LIN {X 0,Y 514.55,Z 869.976,A -85,B 0,C 180,E1 14915.309,E2 14915.309} C_VEL
LIN {X 0,Y 492.785,Z 832.233,A -85,B 0,C 180,E1 14922.914,E2 14922.914} C_VEL
LIN {X 0,Y 477.304,Z 810.224,A -85,B 0,C 180,E1 14930.14,E2 14930.14} C_VEL
LIN {X 0,Y 468.627,Z 798.013,A -85,B 0,C 180,E1 14937.192,E2 14937.192} C_VEL
LIN {X 0,Y 469.402,Z 798.715,A -85,B 0,C 180,E1 14950.485,E2 14950.485} C_VEL
LIN {X 0,Y 482.559,Z 818.186,A -85,B 0,C 180,E1 14959.5,E2 14959.5} C_VEL
LIN {X 0,Y 502.665,Z 847.975,A -85,B 0,C 180,E1 14967.396,E2 14967.396} C_VEL
LIN {X 0,Y 523.166,Z 888.461,A -85,B 0,C 180,E1 14974.072,E2 14974.072} C_VEL
LIN {X 0,Y 527.877,Z 903.855,A -85,B 0,C 180,E1 14975.873,E2 14975.873} C_VEL
LIN {X 0,Y 512.114,Z 972.966,A -85,B 0,C 180,E1 14979.163,E2 14979.163} C_VEL
LIN {X 0,Y 492.159,Z 1039.607,A -85,B 0,C 180,E1 14984.274,E2 14984.274} C_VEL
LIN {X 0,Y 472.146,Z 1098.486,A -85,B 0,C 180,E1 14991.255,E2 14991.255} C_VEL
LIN {X 0,Y 456.172,Z 1146.776,A -85,B 0,C 180,E1 14999.951,E2 14999.951} C_VEL
LIN {X 0,Y 446.7,Z 1181.826,A -85,B 0,C 180,E1 15009.677,E2 15009.677} C_VEL
LIN {X 0,Y 443.594,Z 1200.387,A -85,B 0,C 180,E1 15018.207,E2 15018.207} C_VEL
LIN {X 0,Y 443.244,Z 1209.25,A -85,B 0,C 180,E1 15027.105,E2 15027.105} C_VEL
LIN {X 0,Y 443.109,Z 1207.059,A -85,B 0,C 180,E1 15036.281,E2 15036.281} C_VEL
LIN {X 0,Y 443.626,Z 1202.099,A -85,B 0,C 180,E1 15040.69,E2 15040.69} C_VEL
LIN {X 0,Y 436.653,Z 1194.823,A -85,B 0,C 180,E1 15045.123,E2 15045.123} C_VEL
LIN {X 0,Y 442.918,Z 1167.046,A -85,B 0,C 180,E1 15055.407,E2 15055.407} C_VEL
LIN {X 0,Y 455.683,Z 1125.539,A -85,B 0,C 180,E1 15064.822,E2 15064.822} C_VEL
LIN {X 0,Y 473.88,Z 1072.19,A -85,B 0,C 180,E1 15072.665,E2 15072.665} C_VEL
LIN {X 0,Y 493.668,Z 1009.04,A -85,B 0,C 180,E1 15078.748,E2 15078.748} C_VEL
LIN {X 0,Y 512.086,Z 936.922,A -85,B 0,C 180,E1 15083.109,E2 15083.109} C_VEL
LIN {X 0,Y 518.041,Z 902.964,A -85,B 0,C 180,E1 15084.593,E2 15084.593} C_VEL
LIN {X 0,Y 491.056,Z 847.52,A -85,B 0,C 180,E1 15092.061,E2 15092.061} C_VEL
LIN {X 0,Y 465.874,Z 809.438,A -85,B 0,C 180,E1 15099.537,E2 15099.537} C_VEL
LIN {X 0,Y 445.387,Z 782.11,A -85,B 0,C 180,E1 15108.144,E2 15108.144} C_VEL
LIN {X 0,Y 438.046,Z 773.763,A -85,B 0,C 180,E1 15112.94,E2 15112.94} C_VEL
LIN {X 0,Y 434.63,Z 767.06,A -85,B 0,C 180,E1 15117.025,E2 15117.025} C_VEL
LIN {X 0,Y 434.603,Z 767.06,A -85,B 0,C 180,E1 15127.044,E2 15127.044} C_VEL
LIN {X 0,Y 434.587,Z 769.596,A -85,B 0,C 180,E1 15130.777,E2 15130.777} C_VEL
LIN {X 0,Y 441.296,Z 778.041,A -85,B 0,C 180,E1 15136.565,E2 15136.565} C_VEL
LIN {X 0,Y 453.228,Z 793.03,A -85,B 0,C 180,E1 15142.813,E2 15142.813} C_VEL
LIN {X 0,Y 476.279,Z 824.499,A -85,B 0,C 180,E1 15150.896,E2 15150.896} C_VEL
LIN {X 0,Y 501.922,Z 869.101,A -85,B 0,C 180,E1 15158.245,E2 15158.245} C_VEL
LIN {X 0,Y 517.004,Z 906.387,A -85,B 0,C 180,E1 15162.841,E2 15162.841} C_VEL
LIN {X 0,Y 500.153,Z 980.626,A -85,B 0,C 180,E1 15166.741,E2 15166.741} C_VEL
LIN {X 0,Y 480.671,Z 1045.404,A -85,B 0,C 180,E1 15172.189,E2 15172.189} C_VEL
LIN {X 0,Y 461.137,Z 1102.24,A -85,B 0,C 180,E1 15179.556,E2 15179.556} C_VEL
LIN {X 0,Y 446.003,Z 1147.052,A -85,B 0,C 180,E1 15188.497,E2 15188.497} C_VEL
LIN {X 0,Y 438.075,Z 1177.151,A -85,B 0,C 180,E1 15197.956,E2 15197.956} C_VEL
LIN {X 0,Y 435.754,Z 1194.997,A -85,B 0,C 180,E1 15207.955,E2 15207.955} C_VEL
LIN {X 0,Y 434.823,Z 1200.244,A -85,B 0,C 180,E1 15216.965,E2 15216.965} C_VEL
LIN {X 0,Y 435.396,Z 1194.315,A -85,B 0,C 180,E1 15226.549,E2 15226.549} C_VEL
LIN {X 0,Y 438.157,Z 1176.862,A -85,B 0,C 180,E1 15236.071,E2 15236.071} C_VEL
LIN {X 0,Y 446.753,Z 1145.298,A -85,B 0,C 180,E1 15245.895,E2 15245.895} C_VEL
LIN {X 0,Y 462.863,Z 1099.022,A -85,B 0,C 180,E1 15255.059,E2 15255.059} C_VEL
LIN {X 0,Y 484.058,Z 1040.692,A -85,B 0,C 180,E1 15262.524,E2 15262.524} C_VEL
LIN {X 0,Y 504.988,Z 975.634,A -85,B 0,C 180,E1 15267.875,E2 15267.875} C_VEL
LIN {X 0,Y 521.46,Z 903.347,A -85,B 0,C 180,E1 15271.757,E2 15271.757} C_VEL
LIN {X 0,Y 504.014,Z 862.678,A -85,B 0,C 180,E1 15278.05,E2 15278.05} C_VEL
LIN {X 0,Y 482.677,Z 826.981,A -85,B 0,C 180,E1 15286.689,E2 15286.689} C_VEL
LIN {X 0,Y 471.37,Z 812.429,A -85,B 0,C 180,E1 15293.352,E2 15293.352} C_VEL
LIN {X 0,Y 466.641,Z 805.604,A -85,B 0,C 180,E1 15298.473,E2 15298.473} C_VEL
LIN {X 0,Y 468.304,Z 806.975,A -85,B 0,C 180,E1 15310.415,E2 15310.415} C_VEL
LIN {X 0,Y 480.553,Z 825.384,A -85,B 0,C 180,E1 15319.13,E2 15319.13} C_VEL
LIN {X 0,Y 500.058,Z 855.303,A -85,B 0,C 180,E1 15327.161,E2 15327.161} C_VEL
LIN {X 0,Y 519.378,Z 895.393,A -85,B 0,C 180,E1 15333.839,E2 15333.839} C_VEL
LIN {X 0,Y 522.432,Z 908.933,A -85,B 0,C 180,E1 15335.312,E2 15335.312} C_VEL
LIN {X 0,Y 504.887,Z 981.045,A -85,B 0,C 180,E1 15338.924,E2 15338.924} C_VEL
LIN {X 0,Y 483.99,Z 1046.888,A -85,B 0,C 180,E1 15344.271,E2 15344.271} C_VEL
LIN {X 0,Y 463.175,Z 1105.249,A -85,B 0,C 180,E1 15351.62,E2 15351.62} C_VEL
LIN {X 0,Y 447.239,Z 1151.808,A -85,B 0,C 180,E1 15360.588,E2 15360.588} C_VEL
LIN {X 0,Y 438.359,Z 1184.435,A -85,B 0,C 180,E1 15370.329,E2 15370.329} C_VEL
LIN {X 0,Y 435.527,Z 1203.211,A -85,B 0,C 180,E1 15380.019,E2 15380.019} C_VEL
LIN {X 0,Y 434.847,Z 1209.603,A -85,B 0,C 180,E1 15389.05,E2 15389.05} C_VEL
LIN {X 0,Y 435.31,Z 1205.545,A -85,B 0,C 180,E1 15398.064,E2 15398.064} C_VEL
LIN {X 0,Y 436.653,Z 1194.823,A -85,B 0,C 180,E1 15405.123,E2 15405.123} C_VEL
LIN {X 0,Y 430.369,Z 1185.528,A -85,B 0,C 180,E1 15409.593,E2 15409.593} C_VEL
LIN {X 0,Y 438.934,Z 1154.358,A -85,B 0,C 180,E1 15419.282,E2 15419.282} C_VEL
LIN {X 0,Y 454.389,Z 1109.269,A -85,B 0,C 180,E1 15428.211,E2 15428.211} C_VEL
LIN {X 0,Y 474.785,Z 1051.107,A -85,B 0,C 180,E1 15435.677,E2 15435.677} C_VEL
LIN {X 0,Y 495.141,Z 985.173,A -85,B 0,C 180,E1 15441.123,E2 15441.123} C_VEL
LIN {X 0,Y 512.3,Z 910.236,A -85,B 0,C 180,E1 15444.97,E2 15444.97} C_VEL
LIN {X 0,Y 493.835,Z 865.668,A -85,B 0,C 180,E1 15450.627,E2 15450.627} C_VEL
LIN {X 0,Y 468.539,Z 823.265,A -85,B 0,C 180,E1 15458.23,E2 15458.23} C_VEL
LIN {X 0,Y 447.89,Z 795.765,A -85,B 0,C 180,E1 15466.249,E2 15466.249} C_VEL
LIN {X 0,Y 437.393,Z 781.948,A -85,B 0,C 180,E1 15472.679,E2 15472.679} C_VEL
LIN {X 0,Y 431.938,Z 774.345,A -85,B 0,C 180,E1 15479.02,E2 15479.02} C_VEL
LIN {X 0,Y 433.334,Z 777.105,A -85,B 0,C 180,E1 15490.426,E2 15490.426} C_VEL
LIN {X 0,Y 440.229,Z 786.376,A -85,B 0,C 180,E1 15496.557,E2 15496.557} C_VEL
LIN {X 0,Y 452.443,Z 801.876,A -85,B 0,C 180,E1 15502.948,E2 15502.948} C_VEL
LIN {X 0,Y 474.79,Z 833.633,A -85,B 0,C 180,E1 15510.961,E2 15510.961} C_VEL
LIN {X 0,Y 498.802,Z 877.302,A -85,B 0,C 180,E1 15518.197,E2 15518.197} C_VEL
LIN {X 0,Y 511.362,Z 909.677,A -85,B 0,C 180,E1 15522.262,E2 15522.262} C_VEL
LIN {X 0,Y 493.764,Z 983.834,A -85,B 0,C 180,E1 15526.251,E2 15526.251} C_VEL
LIN {X 0,Y 473.457,Z 1048.85,A -85,B 0,C 180,E1 15531.881,E2 15531.881} C_VEL
LIN {X 0,Y 453.145,Z 1105.724,A -85,B 0,C 180,E1 15539.519,E2 15539.519} C_VEL
LIN {X 0,Y 437.884,Z 1149.454,A -85,B 0,C 180,E1 15548.612,E2 15548.612} C_VEL
LIN {X 0,Y 430.013,Z 1178.764,A -85,B 0,C 180,E1 15558.243,E2 15558.243} C_VEL
LIN {X 0,Y 427.755,Z 1195.235,A -85,B 0,C 180,E1 15567.917,E2 15567.917} C_VEL
LIN {X 0,Y 426.799,Z 1200.316,A -85,B 0,C 180,E1 15577.097,E2 15577.097} C_VEL
LIN {X 0,Y 427.421,Z 1194.277,A -85,B 0,C 180,E1 15586.833,E2 15586.833} C_VEL
LIN {X 0,Y 430.461,Z 1176.392,A -85,B 0,C 180,E1 15596.65,E2 15596.65} C_VEL
LIN {X 0,Y 439.746,Z 1144.653,A -85,B 0,C 180,E1 15606.622,E2 15606.622} C_VEL
LIN {X 0,Y 456.596,Z 1098.752,A -85,B 0,C 180,E1 15615.792,E2 15615.792} C_VEL
LIN {X 0,Y 478.774,Z 1039.962,A -85,B 0,C 180,E1 15623.347,E2 15623.347} C_VEL
LIN {X 0,Y 500.389,Z 974.77,A -85,B 0,C 180,E1 15628.691,E2 15628.691} C_VEL
LIN {X 0,Y 516.503,Z 907.655,A -85,B 0,C 180,E1 15632.309,E2 15632.309} C_VEL
LIN {X 0,Y 500.028,Z 868.149,A -85,B 0,C 180,E1 15638.65,E2 15638.65} C_VEL
LIN {X 0,Y 480.223,Z 834.002,A -85,B 0,C 180,E1 15647.143,E2 15647.143} C_VEL
LIN {X 0,Y 469.728,Z 819.902,A -85,B 0,C 180,E1 15653.718,E2 15653.718} C_VEL
LIN {X 0,Y 465.416,Z 813.419,A -85,B 0,C 180,E1 15658.755,E2 15658.755} C_VEL
LIN {X 0,Y 467.129,Z 815.063,A -85,B 0,C 180,E1 15670.323,E2 15670.323} C_VEL
LIN {X 0,Y 480.744,Z 835.127,A -85,B 0,C 180,E1 15679.859,E2 15679.859} C_VEL
LIN {X 0,Y 500.912,Z 869.272,A -85,B 0,C 180,E1 15688.277,E2 15688.277} C_VEL
LIN {X 0,Y 517.784,Z 909.133,A -85,B 0,C 180,E1 15694.527,E2 15694.527} C_VEL
LIN {X 0,Y 499.734,Z 981.942,A -85,B 0,C 180,E1 15698.228,E2 15698.228} C_VEL
LIN {X 0,Y 478.153,Z 1047.547,A -85,B 0,C 180,E1 15703.603,E2 15703.603} C_VEL
LIN {X 0,Y 456.576,Z 1105.602,A -85,B 0,C 180,E1 15711.004,E2 15711.004} C_VEL
LIN {X 0,Y 439.634,Z 1152.897,A -85,B 0,C 180,E1 15720.313,E2 15720.313} C_VEL
LIN {X 0,Y 430.551,Z 1184.493,A -85,B 0,C 180,E1 15730.018,E2 15730.018} C_VEL
LIN {X 0,Y 427.551,Z 1203.12,A -85,B 0,C 180,E1 15739.83,E2 15739.83} C_VEL
LIN {X 0,Y 426.873,Z 1209.515,A -85,B 0,C 180,E1 15749.032,E2 15749.032} C_VEL
LIN {X 0,Y 427.337,Z 1205.457,A -85,B 0,C 180,E1 15758.215,E2 15758.215} C_VEL
LIN {X 0,Y 429.941,Z 1188.014,A -85,B 0,C 180,E1 15768.571,E2 15768.571} C_VEL
LIN {X 0,Y 430.369,Z 1185.528,A -85,B 0,C 180,E1 15769.593,E2 15769.593} C_VEL
LIN {X 0,Y 425.856,Z 1174.176,A -85,B 0,C 180,E1 15774.06,E2 15774.06} C_VEL
LIN {X 0,Y 438.332,Z 1135.606,A -85,B 0,C 180,E1 15783.994,E2 15783.994} C_VEL
LIN {X 0,Y 456.853,Z 1084.729,A -85,B 0,C 180,E1 15792.4,E2 15792.4} C_VEL
LIN {X 0,Y 478.073,Z 1023.361,A -85,B 0,C 180,E1 15798.975,E2 15798.975} C_VEL
LIN {X 0,Y 498.276,Z 952.795,A -85,B 0,C 180,E1 15803.744,E2 15803.744} C_VEL
LIN {X 0,Y 506.475,Z 909.417,A -85,B 0,C 180,E1 15805.885,E2 15805.885} C_VEL
LIN {X 0,Y 482.175,Z 856.992,A -85,B 0,C 180,E1 15813.391,E2 15813.391} C_VEL
LIN {X 0,Y 458.927,Z 820.13,A -85,B 0,C 180,E1 15821.113,E2 15821.113} C_VEL
LIN {X 0,Y 441.511,Z 796.848,A -85,B 0,C 180,E1 15829.134,E2 15829.134} C_VEL
LIN {X 0,Y 434.885,Z 788.82,A -85,B 0,C 180,E1 15833.894,E2 15833.894} C_VEL
LIN {X 0,Y 430.96,Z 782.28,A -85,B 0,C 180,E1 15839.018,E2 15839.018} C_VEL
LIN {X 0,Y 432.191,Z 784.869,A -85,B 0,C 180,E1 15850.22,E2 15850.22} C_VEL
LIN {X 0,Y 439.245,Z 794.695,A -85,B 0,C 180,E1 15856.595,E2 15856.595} C_VEL
LIN {X 0,Y 453.822,Z 813.27,A -85,B 0,C 180,E1 15864.002,E2 15864.002} C_VEL
LIN {X 0,Y 477.442,Z 849.483,A -85,B 0,C 180,E1 15872.385,E2 15872.385} C_VEL
LIN {X 0,Y 500.408,Z 897.193,A -85,B 0,C 180,E1 15879.731,E2 15879.731} C_VEL
LIN {X 0,Y 505.504,Z 914.613,A -85,B 0,C 180,E1 15881.751,E2 15881.751} C_VEL
LIN {X 0,Y 486.999,Z 988.588,A -85,B 0,C 180,E1 15885.863,E2 15885.863} C_VEL
LIN {X 0,Y 465.562,Z 1054.191,A -85,B 0,C 180,E1 15891.775,E2 15891.775} C_VEL
LIN {X 0,Y 445.179,Z 1109.194,A -85,B 0,C 180,E1 15899.482,E2 15899.482} C_VEL
LIN {X 0,Y 429.819,Z 1151.673,A -85,B 0,C 180,E1 15908.685,E2 15908.685} C_VEL
LIN {X 0,Y 421.865,Z 1181.35,A -85,B 0,C 180,E1 15919.064,E2 15919.064} C_VEL
LIN {X 0,Y 419.252,Z 1196.572,A -85,B 0,C 180,E1 15928.912,E2 15928.912} C_VEL
LIN {X 0,Y 418.788,Z 1200.382,A -85,B 0,C 180,E1 15937.233,E2 15937.233} C_VEL
LIN {X 0,Y 419.384,Z 1194.999,A -85,B 0,C 180,E1 15946.463,E2 15946.463} C_VEL
LIN {X 0,Y 422.481,Z 1177.526,A -85,B 0,C 180,E1 15956.617,E2 15956.617} C_VEL
LIN {X 0,Y 431.699,Z 1147.155,A -85,B 0,C 180,E1 15966.587,E2 15966.587} C_VEL
LIN {X 0,Y 449.506,Z 1100.749,A -85,B 0,C 180,E1 15976.191,E2 15976.191} C_VEL
LIN {X 0,Y 472.404,Z 1042.569,A -85,B 0,C 180,E1 15983.847,E2 15983.847} C_VEL
LIN {X 0,Y 494.981,Z 977.065,A -85,B 0,C 180,E1 15989.32,E2 15989.32} C_VEL
LIN {X 0,Y 511.543,Z 911.986,A -85,B 0,C 180,E1 15992.85,E2 15992.85} C_VEL
LIN {X 0,Y 495.569,Z 872.648,A -85,B 0,C 180,E1 15999.404,E2 15999.404} C_VEL
LIN {X 0,Y 477.405,Z 840.486,A -85,B 0,C 180,E1 16007.765,E2 16007.765} C_VEL
LIN {X 0,Y 468.016,Z 827.308,A -85,B 0,C 180,E1 16014.162,E2 16014.162} C_VEL
LIN {X 0,Y 464.087,Z 821.241,A -85,B 0,C 180,E1 16019.039,E2 16019.039} C_VEL
LIN {X 0,Y 465.855,Z 823.099,A -85,B 0,C 180,E1 16030.233,E2 16030.233} C_VEL
LIN {X 0,Y 478.613,Z 842.662,A -85,B 0,C 180,E1 16039.615,E2 16039.615} C_VEL
LIN {X 0,Y 497.839,Z 876.354,A -85,B 0,C 180,E1 16048.034,E2 16048.034} C_VEL
LIN {X 0,Y 512.649,Z 914.178,A -85,B 0,C 180,E1 16053.989,E2 16053.989} C_VEL
LIN {X 0,Y 494.012,Z 985.118,A -85,B 0,C 180,E1 16057.663,E2 16057.663} C_VEL
LIN {X 0,Y 471.55,Z 1050.512,A -85,B 0,C 180,E1 16063.151,E2 16063.151} C_VEL
LIN {X 0,Y 449.025,Z 1108.65,A -85,B 0,C 180,E1 16070.793,E2 16070.793} C_VEL
LIN {X 0,Y 431.64,Z 1155.035,A -85,B 0,C 180,E1 16080.288,E2 16080.288} C_VEL
LIN {X 0,Y 422.495,Z 1185.621,A -85,B 0,C 180,E1 16090.106,E2 16090.106} C_VEL
LIN {X 0,Y 419.566,Z 1203.029,A -85,B 0,C 180,E1 16099.635,E2 16099.635} C_VEL
LIN {X 0,Y 418.876,Z 1209.427,A -85,B 0,C 180,E1 16109.013,E2 16109.013} C_VEL
LIN {X 0,Y 419.355,Z 1205.369,A -85,B 0,C 180,E1 16118.373,E2 16118.373} C_VEL
LIN {X 0,Y 422.108,Z 1187.915,A -85,B 0,C 180,E1 16128.929,E2 16128.929} C_VEL
LIN {X 0,Y 425.856,Z 1174.176,A -85,B 0,C 180,E1 16134.06,E2 16134.06} C_VEL
LIN {X 0,Y 421.862,Z 1161.045,A -85,B 0,C 180,E1 16138.49,E2 16138.49} C_VEL
LIN {X 0,Y 437.562,Z 1118.086,A -85,B 0,C 180,E1 16147.95,E2 16147.95} C_VEL
LIN {X 0,Y 458.912,Z 1061.878,A -85,B 0,C 180,E1 16155.89,E2 16155.89} C_VEL
LIN {X 0,Y 480.989,Z 996.406,A -85,B 0,C 180,E1 16161.799,E2 16161.799} C_VEL
LIN {X 0,Y 499.946,Z 922.689,A -85,B 0,C 180,E1 16165.927,E2 16165.927} C_VEL
LIN {X 0,Y 500.967,Z 913.275,A -85,B 0,C 180,E1 16166.474,E2 16166.474} C_VEL
LIN {X 0,Y 477.706,Z 861.591,A -85,B 0,C 180,E1 16174.074,E2 16174.074} C_VEL
LIN {X 0,Y 455.273,Z 825.306,A -85,B 0,C 180,E1 16182.013,E2 16182.013} C_VEL
LIN {X 0,Y 438.929,Z 803.289,A -85,B 0,C 180,E1 16190.076,E2 16190.076} C_VEL
LIN {X 0,Y 432.716,Z 795.655,A -85,B 0,C 180,E1 16194.999,E2 16194.999} C_VEL
LIN {X 0,Y 429.98,Z 790.221,A -85,B 0,C 180,E1 16199.016,E2 16199.016} C_VEL
LIN {X 0,Y 431.093,Z 792.782,A -85,B 0,C 180,E1 16210.08,E2 16210.08} C_VEL
LIN {X 0,Y 438.328,Z 803.017,A -85,B 0,C 180,E1 16216.671,E2 16216.671} C_VEL
LIN {X 0,Y 453.039,Z 822.801,A -85,B 0,C 180,E1 16224.244,E2 16224.244} C_VEL
LIN {X 0,Y 474.806,Z 857.596,A -85,B 0,C 180,E1 16232.288,E2 16232.288} C_VEL
LIN {X 0,Y 496.835,Z 905.46,A -85,B 0,C 180,E1 16239.705,E2 16239.705} C_VEL
LIN {X 0,Y 499.853,Z 918.526,A -85,B 0,C 180,E1 16241.179,E2 16241.179} C_VEL
LIN {X 0,Y 480.884,Z 991.174,A -85,B 0,C 180,E1 16245.309,E2 16245.309} C_VEL
LIN {X 0,Y 459.225,Z 1055.188,A -85,B 0,C 180,E1 16251.174,E2 16251.174} C_VEL
LIN {X 0,Y 438.239,Z 1109.828,A -85,B 0,C 180,E1 16258.945,E2 16258.945} C_VEL
LIN {X 0,Y 421.977,Z 1153.148,A -85,B 0,C 180,E1 16268.559,E2 16268.559} C_VEL
LIN {X 0,Y 413.815,Z 1182.819,A -85,B 0,C 180,E1 16279.384,E2 16279.384} C_VEL
LIN {X 0,Y 411.262,Z 1196.763,A -85,B 0,C 180,E1 16288.891,E2 16288.891} C_VEL
LIN {X 0,Y 410.763,Z 1200.448,A -85,B 0,C 180,E1 16297.376,E2 16297.376} C_VEL
LIN {X 0,Y 411.403,Z 1194.925,A -85,B 0,C 180,E1 16306.792,E2 16306.792} C_VEL
LIN {X 0,Y 414.813,Z 1177.3,A -85,B 0,C 180,E1 16317.149,E2 16317.149} C_VEL
LIN {X 0,Y 425.203,Z 1145.596,A -85,B 0,C 180,E1 16327.604,E2 16327.604} C_VEL
LIN {X 0,Y 444.044,Z 1098.944,A -85,B 0,C 180,E1 16337.206,E2 16337.206} C_VEL
LIN {X 0,Y 467.642,Z 1040.906,A -85,B 0,C 180,E1 16344.804,E2 16344.804} C_VEL
LIN {X 0,Y 490.845,Z 975.353,A -85,B 0,C 180,E1 16350.219,E2 16350.219} C_VEL
LIN {X 0,Y 506.305,Z 915.237,A -85,B 0,C 180,E1 16353.557,E2 16353.557} C_VEL
LIN {X 0,Y 490.777,Z 876.376,A -85,B 0,C 180,E1 16360.346,E2 16360.346} C_VEL
LIN {X 0,Y 472.953,Z 843.336,A -85,B 0,C 180,E1 16369.507,E2 16369.507} C_VEL
LIN {X 0,Y 463.277,Z 829.372,A -85,B 0,C 180,E1 16378.462,E2 16378.462} C_VEL
LIN {X 0,Y 464.478,Z 830.678,A -85,B 0,C 180,E1 16389.967,E2 16389.967} C_VEL
LIN {X 0,Y 476.611,Z 850.351,A -85,B 0,C 180,E1 16399.43,E2 16399.43} C_VEL
LIN {X 0,Y 494.619,Z 883.467,A -85,B 0,C 180,E1 16407.801,E2 16407.801} C_VEL
LIN {X 0,Y 507.427,Z 918.393,A -85,B 0,C 180,E1 16413.381,E2 16413.381} C_VEL
LIN {X 0,Y 488.169,Z 988.544,A -85,B 0,C 180,E1 16417.116,E2 16417.116} C_VEL
LIN {X 0,Y 464.609,Z 1054.247,A -85,B 0,C 180,E1 16422.779,E2 16422.779} C_VEL
LIN {X 0,Y 441.315,Z 1111.762,A -85,B 0,C 180,E1 16430.619,E2 16430.619} C_VEL
LIN {X 0,Y 424.023,Z 1156.032,A -85,B 0,C 180,E1 16439.995,E2 16439.995} C_VEL
LIN {X 0,Y 414.428,Z 1186.908,A -85,B 0,C 180,E1 16450.26,E2 16450.26} C_VEL
LIN {X 0,Y 411.513,Z 1204.166,A -85,B 0,C 180,E1 16460.502,E2 16460.502} C_VEL
LIN {X 0,Y 410.884,Z 1209.34,A -85,B 0,C 180,E1 16468.994,E2 16468.994} C_VEL
LIN {X 0,Y 411.376,Z 1205.281,A -85,B 0,C 180,E1 16478.537,E2 16478.537} C_VEL
LIN {X 0,Y 414.049,Z 1188.962,A -85,B 0,C 180,E1 16488.756,E2 16488.756} C_VEL
LIN {X 0,Y 421.862,Z 1161.045,A -85,B 0,C 180,E1 16498.49,E2 16498.49} C_VEL
LIN {X 0,Y 420.256,Z 1145.942,A -85,B 0,C 180,E1 16502.86,E2 16502.86} C_VEL
LIN {X 0,Y 439.337,Z 1097.118,A -85,B 0,C 180,E1 16512.009,E2 16512.009} C_VEL
LIN {X 0,Y 462.147,Z 1036.978,A -85,B 0,C 180,E1 16519.205,E2 16519.205} C_VEL
LIN {X 0,Y 484.206,Z 968.139,A -85,B 0,C 180,E1 16524.369,E2 16524.369} C_VEL
LIN {X 0,Y 495.541,Z 917.435,A -85,B 0,C 180,E1 16527.016,E2 16527.016} C_VEL
LIN {X 0,Y 473.775,Z 867.125,A -85,B 0,C 180,E1 16534.607,E2 16534.607} C_VEL
LIN {X 0,Y 452.648,Z 831.996,A -85,B 0,C 180,E1 16542.535,E2 16542.535} C_VEL
LIN {X 0,Y 436.417,Z 809.309,A -85,B 0,C 180,E1 16551.091,E2 16551.091} C_VEL
LIN {X 0,Y 429,Z 798.169,A -85,B 0,C 180,E1 16559.014,E2 16559.014} C_VEL
LIN {X 0,Y 430.043,Z 800.853,A -85,B 0,C 180,E1 16570.02,E2 16570.02} C_VEL
LIN {X 0,Y 440.022,Z 813.855,A -85,B 0,C 180,E1 16578.36,E2 16578.36} C_VEL
LIN {X 0,Y 459.198,Z 842.928,A -85,B 0,C 180,E1 16587.391,E2 16587.391} C_VEL
LIN {X 0,Y 480.77,Z 883.187,A -85,B 0,C 180,E1 16595.229,E2 16595.229} C_VEL
LIN {X 0,Y 494.47,Z 921.548,A -85,B 0,C 180,E1 16600.56,E2 16600.56} C_VEL
LIN {X 0,Y 474.387,Z 995.114,A -85,B 0,C 180,E1 16604.836,E2 16604.836} C_VEL
LIN {X 0,Y 451.566,Z 1059.945,A -85,B 0,C 180,E1 16610.99,E2 16610.99} C_VEL
LIN {X 0,Y 429.74,Z 1114.637,A -85,B 0,C 180,E1 16619.148,E2 16619.148} C_VEL
LIN {X 0,Y 413.578,Z 1156.494,A -85,B 0,C 180,E1 16628.986,E2 16628.986} C_VEL
LIN {X 0,Y 405.728,Z 1184.272,A -85,B 0,C 180,E1 16639.714,E2 16639.714} C_VEL
LIN {X 0,Y 403.265,Z 1196.954,A -85,B 0,C 180,E1 16648.869,E2 16648.869} C_VEL
LIN {X 0,Y 402.738,Z 1200.514,A -85,B 0,C 180,E1 16657.523,E2 16657.523} C_VEL
LIN {X 0,Y 403.482,Z 1194.519,A -85,B 0,C 180,E1 16667.451,E2 16667.451} C_VEL
LIN {X 0,Y 407.213,Z 1177.09,A -85,B 0,C 180,E1 16677.699,E2 16677.699} C_VEL
LIN {X 0,Y 418.436,Z 1144.961,A -85,B 0,C 180,E1 16688.404,E2 16688.404} C_VEL
LIN {X 0,Y 438.123,Z 1098.419,A -85,B 0,C 180,E1 16698.049,E2 16698.049} C_VEL
LIN {X 0,Y 462.683,Z 1040.203,A -85,B 0,C 180,E1 16705.677,E2 16705.677} C_VEL
LIN {X 0,Y 486.485,Z 974.705,A -85,B 0,C 180,E1 16711.071,E2 16711.071} C_VEL
LIN {X 0,Y 501.146,Z 918.658,A -85,B 0,C 180,E1 16714.266,E2 16714.266} C_VEL
LIN {X 0,Y 486.106,Z 880.111,A -85,B 0,C 180,E1 16721.313,E2 16721.313} C_VEL
LIN {X 0,Y 470.211,Z 850.206,A -85,B 0,C 180,E1 16730.173,E2 16730.173} C_VEL
LIN {X 0,Y 461.635,Z 837.117,A -85,B 0,C 180,E1 16738.745,E2 16738.745} C_VEL
LIN {X 0,Y 462.92,Z 838.769,A -85,B 0,C 180,E1 16749.941,E2 16749.941} C_VEL
LIN {X 0,Y 474.261,Z 857.796,A -85,B 0,C 180,E1 16759.19,E2 16759.19} C_VEL
LIN {X 0,Y 491.15,Z 890.074,A -85,B 0,C 180,E1 16767.459,E2 16767.459} C_VEL
LIN {X 0,Y 502.417,Z 921.829,A -85,B 0,C 180,E1 16772.72,E2 16772.72} C_VEL
LIN {X 0,Y 481.821,Z 993.409,A -85,B 0,C 180,E1 16776.657,E2 16776.657} C_VEL
LIN {X 0,Y 457.352,Z 1058.574,A -85,B 0,C 180,E1 16782.477,E2 16782.477} C_VEL
LIN {X 0,Y 433.299,Z 1115.503,A -85,B 0,C 180,E1 16790.556,E2 16790.556} C_VEL
LIN {X 0,Y 415.332,Z 1159.961,A -85,B 0,C 180,E1 16800.51,E2 16800.51} C_VEL
LIN {X 0,Y 406.091,Z 1189.183,A -85,B 0,C 180,E1 16810.974,E2 16810.974} C_VEL
LIN {X 0,Y 403.482,Z 1205.285,A -85,B 0,C 180,E1 16821.403,E2 16821.403} C_VEL
LIN {X 0,Y 402.886,Z 1209.252,A -85,B 0,C 180,E1 16828.974,E2 16828.974} C_VEL
LIN {X 0,Y 403.41,Z 1205.188,A -85,B 0,C 180,E1 16838.706,E2 16838.706} C_VEL
LIN {X 0,Y 406.213,Z 1188.829,A -85,B 0,C 180,E1 16849.132,E2 16849.132} C_VEL
LIN {X 0,Y 414.721,Z 1160.313,A -85,B 0,C 180,E1 16859.186,E2 16859.186} C_VEL
LIN {X 0,Y 420.256,Z 1145.942,A -85,B 0,C 180,E1 16862.86,E2 16862.86} C_VEL
LIN {X 0,Y 419.652,Z 1129.083,A -85,B 0,C 180,E1 16867.132,E2 16867.132} C_VEL
LIN {X 0,Y 441.363,Z 1076.326,A -85,B 0,C 180,E1 16875.575,E2 16875.575} C_VEL
LIN {X 0,Y 464.933,Z 1012.723,A -85,B 0,C 180,E1 16882.076,E2 16882.076} C_VEL
LIN {X 0,Y 486.357,Z 940.377,A -85,B 0,C 180,E1 16886.623,E2 16886.623} C_VEL
LIN {X 0,Y 489.86,Z 920.725,A -85,B 0,C 180,E1 16887.686,E2 16887.686} C_VEL
LIN {X 0,Y 469.225,Z 871.636,A -85,B 0,C 180,E1 16895.366,E2 16895.366} C_VEL
LIN {X 0,Y 449.547,Z 838.208,A -85,B 0,C 180,E1 16903.169,E2 16903.169} C_VEL
LIN {X 0,Y 433.29,Z 813.717,A -85,B 0,C 180,E1 16912.735,E2 16912.735} C_VEL
LIN {X 0,Y 427.507,Z 806.001,A -85,B 0,C 180,E1 16920.027,E2 16920.027} C_VEL
LIN {X 0,Y 428.949,Z 808.729,A -85,B 0,C 180,E1 16929.875,E2 16929.875} C_VEL
LIN {X 0,Y 438.519,Z 821.875,A -85,B 0,C 180,E1 16938.212,E2 16938.212} C_VEL
LIN {X 0,Y 457.02,Z 850.719,A -85,B 0,C 180,E1 16947.26,E2 16947.26} C_VEL
LIN {X 0,Y 477.068,Z 890.155,A -85,B 0,C 180,E1 16954.986,E2 16954.986} C_VEL
LIN {X 0,Y 489.094,Z 924.788,A -85,B 0,C 180,E1 16959.938,E2 16959.938} C_VEL
LIN {X 0,Y 468.62,Z 996.843,A -85,B 0,C 180,E1 16964.194,E2 16964.194} C_VEL
LIN {X 0,Y 445.214,Z 1061.087,A -85,B 0,C 180,E1 16970.384,E2 16970.384} C_VEL
LIN {X 0,Y 422.808,Z 1115.207,A -85,B 0,C 180,E1 16978.585,E2 16978.585} C_VEL
LIN {X 0,Y 406.006,Z 1156.923,A -85,B 0,C 180,E1 16988.575,E2 16988.575} C_VEL
LIN {X 0,Y 397.806,Z 1184.573,A -85,B 0,C 180,E1 16999.507,E2 16999.507} C_VEL
LIN {X 0,Y 395.283,Z 1197.138,A -85,B 0,C 180,E1 17008.846,E2 17008.846} C_VEL
LIN {X 0,Y 394.714,Z 1200.581,A -85,B 0,C 180,E1 17017.677,E2 17017.677} C_VEL
LIN {X 0,Y 395.541,Z 1194.469,A -85,B 0,C 180,E1 17027.814,E2 17027.814} C_VEL
LIN {X 0,Y 399.624,Z 1176.894,A -85,B 0,C 180,E1 17038.272,E2 17038.272} C_VEL
LIN {X 0,Y 411.486,Z 1145.037,A -85,B 0,C 180,E1 17049.048,E2 17049.048} C_VEL
LIN {X 0,Y 432.337,Z 1097.908,A -85,B 0,C 180,E1 17058.909,E2 17058.909} C_VEL
LIN {X 0,Y 457.65,Z 1039.965,A -85,B 0,C 180,E1 17066.523,E2 17066.523} C_VEL
LIN {X 0,Y 481.911,Z 975.24,A -85,B 0,C 180,E1 17071.853,E2 17071.853} C_VEL
LIN {X 0,Y 496.331,Z 923.066,A -85,B 0,C 180,E1 17074.844,E2 17074.844} C_VEL
LIN {X 0,Y 482.002,Z 885.201,A -85,B 0,C 180,E1 17082.046,E2 17082.046} C_VEL
LIN {X 0,Y 467.619,Z 857.331,A -85,B 0,C 180,E1 17090.608,E2 17090.608} C_VEL
LIN {X 0,Y 460.227,Z 845.045,A -85,B 0,C 180,E1 17098.559,E2 17098.559} C_VEL
LIN {X 0,Y 461.25,Z 846.399,A -85,B 0,C 180,E1 17109.738,E2 17109.738} C_VEL
LIN {X 0,Y 471.951,Z 865.484,A -85,B 0,C 180,E1 17119.027,E2 17119.027} C_VEL
LIN {X 0,Y 487.536,Z 896.59,A -85,B 0,C 180,E1 17127.123,E2 17127.123} C_VEL
LIN {X 0,Y 497.118,Z 926.807,A -85,B 0,C 180,E1 17132.112,E2 17132.112} C_VEL
LIN {X 0,Y 475.432,Z 998.631,A -85,B 0,C 180,E1 17136.218,E2 17136.218} C_VEL
LIN {X 0,Y 450.274,Z 1062.598,A -85,B 0,C 180,E1 17142.134,E2 17142.134} C_VEL
LIN {X 0,Y 425.307,Z 1119.19,A -85,B 0,C 180,E1 17150.478,E2 17150.478} C_VEL
LIN {X 0,Y 407.075,Z 1162.625,A -85,B 0,C 180,E1 17160.678,E2 17160.678} C_VEL
LIN {X 0,Y 398.031,Z 1190.303,A -85,B 0,C 180,E1 17171.151,E2 17171.151} C_VEL
LIN {X 0,Y 395.499,Z 1205.208,A -85,B 0,C 180,E1 17181.228,E2 17181.228} C_VEL
LIN {X 0,Y 394.902,Z 1209.167,A -85,B 0,C 180,E1 17188.954,E2 17188.954} C_VEL
LIN {X 0,Y 395.45,Z 1205.085,A -85,B 0,C 180,E1 17198.883,E2 17198.883} C_VEL
LIN {X 0,Y 398.391,Z 1188.685,A -85,B 0,C 180,E1 17209.523,E2 17209.523} C_VEL
LIN {X 0,Y 407.44,Z 1160.051,A -85,B 0,C 180,E1 17219.772,E2 17219.772} C_VEL
LIN {X 0,Y 419.652,Z 1129.083,A -85,B 0,C 180,E1 17227.132,E2 17227.132} C_VEL
LIN {X 0,Y 420.778,Z 1110.521,A -85,B 0,C 180,E1 17231.255,E2 17231.255} C_VEL
LIN {X 0,Y 444.742,Z 1053.025,A -85,B 0,C 180,E1 17239.082,E2 17239.082} C_VEL
LIN {X 0,Y 468.234,Z 987.673,A -85,B 0,C 180,E1 17244.679,E2 17244.679} C_VEL
LIN {X 0,Y 484.349,Z 924.216,A -85,B 0,C 180,E1 17248.338,E2 17248.338} C_VEL
LIN {X 0,Y 464.637,Z 876.026,A -85,B 0,C 180,E1 17256.133,E2 17256.133} C_VEL
LIN {X 0,Y 444.996,Z 841.52,A -85,B 0,C 180,E1 17264.581,E2 17264.581} C_VEL
LIN {X 0,Y 431.205,Z 821.046,A -85,B 0,C 180,E1 17273.462,E2 17273.462} C_VEL
LIN {X 0,Y 426.985,Z 814.023,A -85,B 0,C 180,E1 17279.009,E2 17279.009} C_VEL
LIN {X 0,Y 427.718,Z 816.619,A -85,B 0,C 180,E1 17289.733,E2 17289.733} C_VEL
LIN {X 0,Y 436.979,Z 829.758,A -85,B 0,C 180,E1 17298.037,E2 17298.037} C_VEL
LIN {X 0,Y 454.303,Z 858.065,A -85,B 0,C 180,E1 17307.023,E2 17307.023} C_VEL
LIN {X 0,Y 473.799,Z 898.438,A -85,B 0,C 180,E1 17314.983,E2 17314.983} C_VEL
LIN {X 0,Y 483.507,Z 928.625,A -85,B 0,C 180,E1 17319.343,E2 17319.343} C_VEL
LIN {X 0,Y 462.004,Z 1000.956,A -85,B 0,C 180,E1 17323.736,E2 17323.736} C_VEL
LIN {X 0,Y 437.914,Z 1064.589,A -85,B 0,C 180,E1 17330.071,E2 17330.071} C_VEL
LIN {X 0,Y 415.294,Z 1117.186,A -85,B 0,C 180,E1 17338.289,E2 17338.289} C_VEL
LIN {X 0,Y 398.477,Z 1157.34,A -85,B 0,C 180,E1 17348.149,E2 17348.149} C_VEL
LIN {X 0,Y 390.079,Z 1183.814,A -85,B 0,C 180,E1 17358.729,E2 17358.729} C_VEL
LIN {X 0,Y 387.304,Z 1197.317,A -85,B 0,C 180,E1 17368.822,E2 17368.822} C_VEL
LIN {X 0,Y 386.691,Z 1200.65,A -85,B 0,C 180,E1 17377.837,E2 17377.837} C_VEL
LIN {X 0,Y 387.602,Z 1194.427,A -85,B 0,C 180,E1 17388.192,E2 17388.192} C_VEL
LIN {X 0,Y 392.094,Z 1176.707,A -85,B 0,C 180,E1 17398.865,E2 17398.865} C_VEL
LIN {X 0,Y 405.353,Z 1143.432,A -85,B 0,C 180,E1 17410.153,E2 17410.153} C_VEL
LIN {X 0,Y 427.265,Z 1096.064,A -85,B 0,C 180,E1 17420.015,E2 17420.015} C_VEL
LIN {X 0,Y 453.161,Z 1038.727,A -85,B 0,C 180,E1 17427.488,E2 17427.488} C_VEL
LIN {X 0,Y 478.022,Z 973.965,A -85,B 0,C 180,E1 17432.768,E2 17432.768} C_VEL
LIN {X 0,Y 491.254,Z 926.754,A -85,B 0,C 180,E1 17435.556,E2 17435.556} C_VEL
LIN {X 0,Y 478.499,Z 891.624,A -85,B 0,C 180,E1 17442.447,E2 17442.447} C_VEL
LIN {X 0,Y 465.209,Z 864.568,A -85,B 0,C 180,E1 17450.947,E2 17450.947} C_VEL
LIN {X 0,Y 458.341,Z 852.678,A -85,B 0,C 180,E1 17459.027,E2 17459.027} C_VEL
LIN {X 0,Y 459.55,Z 854.557,A -85,B 0,C 180,E1 17469.774,E2 17469.774} C_VEL
LIN {X 0,Y 469.475,Z 872.784,A -85,B 0,C 180,E1 17478.765,E2 17478.765} C_VEL
LIN {X 0,Y 483.722,Z 902.785,A -85,B 0,C 180,E1 17486.725,E2 17486.725} C_VEL
LIN {X 0,Y 492.098,Z 930.927,A -85,B 0,C 180,E1 17491.459,E2 17491.459} C_VEL
LIN {X 0,Y 468.922,Z 1004.044,A -85,B 0,C 180,E1 17495.781,E2 17495.781} C_VEL
LIN {X 0,Y 442.89,Z 1067.371,A -85,B 0,C 180,E1 17501.87,E2 17501.87} C_VEL
LIN {X 0,Y 417.043,Z 1123.341,A -85,B 0,C 180,E1 17510.522,E2 17510.522} C_VEL
LIN {X 0,Y 398.456,Z 1165.98,A -85,B 0,C 180,E1 17521.139,E2 17521.139} C_VEL
LIN {X 0,Y 389.68,Z 1193.407,A -85,B 0,C 180,E1 17532.407,E2 17532.407} C_VEL
LIN {X 0,Y 387.359,Z 1206.008,A -85,B 0,C 180,E1 17542.176,E2 17542.176} C_VEL
LIN {X 0,Y 386.852,Z 1209.057,A -85,B 0,C 180,E1 17551.179,E2 17551.179} C_VEL
LIN {X 0,Y 387.725,Z 1202.543,A -85,B 0,C 180,E1 17561.316,E2 17561.316} C_VEL
LIN {X 0,Y 391.987,Z 1183.661,A -85,B 0,C 180,E1 17572.112,E2 17572.112} C_VEL
LIN {X 0,Y 404.265,Z 1149.902,A -85,B 0,C 180,E1 17583.034,E2 17583.034} C_VEL
LIN {X 0,Y 420.778,Z 1110.521,A -85,B 0,C 180,E1 17591.255,E2 17591.255} C_VEL
LIN {X 0,Y 423.409,Z 1090.051,A -85,B 0,C 180,E1 17595.183,E2 17595.183} C_VEL
LIN {X 0,Y 448.699,Z 1028.256,A -85,B 0,C 180,E1 17602.303,E2 17602.303} C_VEL
LIN {X 0,Y 472.447,Z 957.337,A -85,B 0,C 180,E1 17607.306,E2 17607.306} C_VEL
LIN {X 0,Y 479.319,Z 929.095,A -85,B 0,C 180,E1 17608.814,E2 17608.814} C_VEL
LIN {X 0,Y 460.615,Z 881.504,A -85,B 0,C 180,E1 17616.688,E2 17616.688} C_VEL
LIN {X 0,Y 442.003,Z 847.969,A -85,B 0,C 180,E1 17625.238,E2 17625.238} C_VEL
LIN {X 0,Y 429.465,Z 828.597,A -85,B 0,C 180,E1 17633.944,E2 17633.944} C_VEL
LIN {X 0,Y 425.83,Z 821.915,A -85,B 0,C 180,E1 17639.006,E2 17639.006} C_VEL
LIN {X 0,Y 426.456,Z 824.454,A -85,B 0,C 180,E1 17649.59,E2 17649.59} C_VEL
LIN {X 0,Y 435.088,Z 837.56,A -85,B 0,C 180,E1 17657.856,E2 17657.856} C_VEL
LIN {X 0,Y 451.403,Z 865.045,A -85,B 0,C 180,E1 17666.696,E2 17666.696} C_VEL
LIN {X 0,Y 469.94,Z 905.366,A -85,B 0,C 180,E1 17674.747,E2 17674.747} C_VEL
LIN {X 0,Y 477.856,Z 932.848,A -85,B 0,C 180,E1 17678.754,E2 17678.754} C_VEL
LIN {X 0,Y 455.453,Z 1004.937,A -85,B 0,C 180,E1 17683.255,E2 17683.255} C_VEL
LIN {X 0,Y 430.167,Z 1069.051,A -85,B 0,C 180,E1 17689.866,E2 17689.866} C_VEL
LIN {X 0,Y 406.76,Z 1121.477,A -85,B 0,C 180,E1 17698.457,E2 17698.457} C_VEL
LIN {X 0,Y 389.576,Z 1161.636,A -85,B 0,C 180,E1 17709.006,E2 17709.006} C_VEL
LIN {X 0,Y 381.189,Z 1187.964,A -85,B 0,C 180,E1 17720.782,E2 17720.782} C_VEL
LIN {X 0,Y 379.049,Z 1199.133,A -85,B 0,C 180,E1 17731.09,E2 17731.09} C_VEL
LIN {X 0,Y 378.675,Z 1200.06,A -85,B 0,C 180,E1 17740.894,E2 17740.894} C_VEL
LIN {X 0,Y 380.329,Z 1191.274,A -85,B 0,C 180,E1 17751.108,E2 17751.108} C_VEL
LIN {X 0,Y 387.794,Z 1168.159,A -85,B 0,C 180,E1 17762.967,E2 17762.967} C_VEL
LIN {X 0,Y 404.702,Z 1130.153,A -85,B 0,C 180,E1 17774.202,E2 17774.202} C_VEL
LIN {X 0,Y 429.36,Z 1079.756,A -85,B 0,C 180,E1 17783.36,E2 17783.36} C_VEL
LIN {X 0,Y 456.444,Z 1019.259,A -85,B 0,C 180,E1 17790.232,E2 17790.232} C_VEL
LIN {X 0,Y 481.722,Z 949.753,A -85,B 0,C 180,E1 17795.039,E2 17795.039} C_VEL
LIN {X 0,Y 486.524,Z 931.857,A -85,B 0,C 180,E1 17796.033,E2 17796.033} C_VEL
LIN {X 0,Y 474.246,Z 896.387,A -85,B 0,C 180,E1 17803.244,E2 17803.244} C_VEL
LIN {X 0,Y 462.603,Z 871.655,A -85,B 0,C 180,E1 17811.371,E2 17811.371} C_VEL
LIN {X 0,Y 456.47,Z 860.462,A -85,B 0,C 180,E1 17819.023,E2 17819.023} C_VEL
LIN {X 0,Y 457.569,Z 862.321,A -85,B 0,C 180,E1 17829.659,E2 17829.659} C_VEL
LIN {X 0,Y 466.791,Z 880.243,A -85,B 0,C 180,E1 17838.569,E2 17838.569} C_VEL
LIN {X 0,Y 480.268,Z 909.855,A -85,B 0,C 180,E1 17846.5,E2 17846.5} C_VEL
LIN {X 0,Y 487.019,Z 934.993,A -85,B 0,C 180,E1 17850.808,E2 17850.808} C_VEL
LIN {X 0,Y 463.114,Z 1007.265,A -85,B 0,C 180,E1 17855.183,E2 17855.183} C_VEL
LIN {X 0,Y 436.477,Z 1069.625,A -85,B 0,C 180,E1 17861.318,E2 17861.318} C_VEL
LIN {X 0,Y 410.594,Z 1123.482,A -85,B 0,C 180,E1 17869.777,E2 17869.777} C_VEL
LIN {X 0,Y 391.363,Z 1165.509,A -85,B 0,C 180,E1 17880.377,E2 17880.377} C_VEL
LIN {X 0,Y 382.079,Z 1191.9,A -85,B 0,C 180,E1 17891.191,E2 17891.191} C_VEL
LIN {X 0,Y 379.373,Z 1205.94,A -85,B 0,C 180,E1 17902.01,E2 17902.01} C_VEL
LIN {X 0,Y 378.878,Z 1208.966,A -85,B 0,C 180,E1 17911.204,E2 17911.204} C_VEL
LIN {X 0,Y 379.61,Z 1203.629,A -85,B 0,C 180,E1 17920.419,E2 17920.419} C_VEL
LIN {X 0,Y 383.421,Z 1186.417,A -85,B 0,C 180,E1 17931.317,E2 17931.317} C_VEL
LIN {X 0,Y 395.078,Z 1154.595,A -85,B 0,C 180,E1 17942.42,E2 17942.42} C_VEL
LIN {X 0,Y 415.279,Z 1108.494,A -85,B 0,C 180,E1 17952.314,E2 17952.314} C_VEL
LIN {X 0,Y 423.409,Z 1090.051,A -85,B 0,C 180,E1 17955.183,E2 17955.183} C_VEL
LIN {X 0,Y 427.088,Z 1068.053,A -85,B 0,C 180,E1 17958.911,E2 17958.911} C_VEL
LIN {X 0,Y 453.079,Z 1002.759,A -85,B 0,C 180,E1 17965.213,E2 17965.213} C_VEL
LIN {X 0,Y 473.606,Z 931.954,A -85,B 0,C 180,E1 17969.591,E2 17969.591} C_VEL
LIN {X 0,Y 456.136,Z 886.115,A -85,B 0,C 180,E1 17977.456,E2 17977.456} C_VEL
LIN {X 0,Y 438.776,Z 854.005,A -85,B 0,C 180,E1 17986.022,E2 17986.022} C_VEL
LIN {X 0,Y 427.56,Z 836.055,A -85,B 0,C 180,E1 17994.428,E2 17994.428} C_VEL
LIN {X 0,Y 424.155,Z 829.735,A -85,B 0,C 180,E1 18000.027,E2 18000.027} C_VEL
LIN {X 0,Y 425.145,Z 832.421,A -85,B 0,C 180,E1 18009.532,E2 18009.532} C_VEL
LIN {X 0,Y 433.292,Z 845.459,A -85,B 0,C 180,E1 18017.735,E2 18017.735} C_VEL
LIN {X 0,Y 448.911,Z 872.897,A -85,B 0,C 180,E1 18026.625,E2 18026.625} C_VEL
LIN {X 0,Y 466.313,Z 913.419,A -85,B 0,C 180,E1 18034.73,E2 18034.73} C_VEL
LIN {X 0,Y 472.372,Z 936.492,A -85,B 0,C 180,E1 18038.119,E2 18038.119} C_VEL
LIN {X 0,Y 449.291,Z 1007.992,A -85,B 0,C 180,E1 18042.689,E2 18042.689} C_VEL
LIN {X 0,Y 424.046,Z 1069.777,A -85,B 0,C 180,E1 18049.165,E2 18049.165} C_VEL
LIN {X 0,Y 399.89,Z 1122.026,A -85,B 0,C 180,E1 18057.851,E2 18057.851} C_VEL
LIN {X 0,Y 381.919,Z 1162.343,A -85,B 0,C 180,E1 18068.672,E2 18068.672} C_VEL
LIN {X 0,Y 373.3,Z 1188.236,A -85,B 0,C 180,E1 18080.585,E2 18080.585} C_VEL
LIN {X 0,Y 371.074,Z 1199.272,A -85,B 0,C 180,E1 18091.114,E2 18091.114} C_VEL
LIN {X 0,Y 370.673,Z 1200.346,A -85,B 0,C 180,E1 18100.556,E2 18100.556} C_VEL
LIN {X 0,Y 372.459,Z 1191.371,A -85,B 0,C 180,E1 18111.446,E2 18111.446} C_VEL
LIN {X 0,Y 380.137,Z 1168.819,A -85,B 0,C 180,E1 18123.342,E2 18123.342} C_VEL
LIN {X 0,Y 397.808,Z 1130.998,A -85,B 0,C 180,E1 18134.802,E2 18134.802} C_VEL
LIN {X 0,Y 423.251,Z 1081.101,A -85,B 0,C 180,E1 18144.033,E2 18144.033} C_VEL
LIN {X 0,Y 451.486,Z 1020.179,A -85,B 0,C 180,E1 18151.031,E2 18151.031} C_VEL
LIN {X 0,Y 477.359,Z 951.2,A -85,B 0,C 180,E1 18155.821,E2 18155.821} C_VEL
LIN {X 0,Y 481.447,Z 935.453,A -85,B 0,C 180,E1 18156.78,E2 18156.78} C_VEL
LIN {X 0,Y 470.05,Z 901.273,A -85,B 0,C 180,E1 18164.054,E2 18164.054} C_VEL
LIN {X 0,Y 459.643,Z 878.26,A -85,B 0,C 180,E1 18171.972,E2 18171.972} C_VEL
LIN {X 0,Y 454.36,Z 868.11,A -85,B 0,C 180,E1 18179.497,E2 18179.497} C_VEL
LIN {X 0,Y 455.637,Z 870.181,A -85,B 0,C 180,E1 18189.621,E2 18189.621} C_VEL
LIN {X 0,Y 464.372,Z 888.152,A -85,B 0,C 180,E1 18198.546,E2 18198.546} C_VEL
LIN {X 0,Y 476.824,Z 917.489,A -85,B 0,C 180,E1 18206.422,E2 18206.422} C_VEL
LIN {X 0,Y 482.04,Z 938.922,A -85,B 0,C 180,E1 18210.138,E2 18210.138} C_VEL
LIN {X 0,Y 457.529,Z 1010.082,A -85,B 0,C 180,E1 18214.54,E2 18214.54} C_VEL
LIN {X 0,Y 430.093,Z 1071.889,A -85,B 0,C 180,E1 18220.747,E2 18220.747} C_VEL
LIN {X 0,Y 402.911,Z 1126.264,A -85,B 0,C 180,E1 18229.56,E2 18229.56} C_VEL
LIN {X 0,Y 383.283,Z 1167.455,A -85,B 0,C 180,E1 18240.406,E2 18240.406} C_VEL
LIN {X 0,Y 373.729,Z 1194.462,A -85,B 0,C 180,E1 18252.333,E2 18252.333} C_VEL
LIN {X 0,Y 371.385,Z 1205.875,A -85,B 0,C 180,E1 18261.837,E2 18261.837} C_VEL
LIN {X 0,Y 370.904,Z 1208.874,A -85,B 0,C 180,E1 18271.23,E2 18271.23} C_VEL
LIN {X 0,Y 371.625,Z 1203.506,A -85,B 0,C 180,E1 18280.646,E2 18280.646} C_VEL
LIN {X 0,Y 376.006,Z 1185.436,A -85,B 0,C 180,E1 18292.124,E2 18292.124} C_VEL
LIN {X 0,Y 388.711,Z 1152.872,A -85,B 0,C 180,E1 18303.472,E2 18303.472} C_VEL
LIN {X 0,Y 410.254,Z 1105.545,A -85,B 0,C 180,E1 18313.526,E2 18313.526} C_VEL
LIN {X 0,Y 427.088,Z 1068.053,A -85,B 0,C 180,E1 18318.911,E2 18318.911} C_VEL
LIN {X 0,Y 431.667,Z 1044.263,A -85,B 0,C 180,E1 18322.373,E2 18322.373} C_VEL
LIN {X 0,Y 456.796,Z 977.636,A -85,B 0,C 180,E1 18327.751,E2 18327.751} C_VEL
LIN {X 0,Y 468.224,Z 935.925,A -85,B 0,C 180,E1 18330.205,E2 18330.205} C_VEL
LIN {X 0,Y 452.062,Z 891.477,A -85,B 0,C 180,E1 18338.085,E2 18338.085} C_VEL
LIN {X 0,Y 435.611,Z 860.096,A -85,B 0,C 180,E1 18346.726,E2 18346.726} C_VEL
LIN {X 0,Y 425.441,Z 843.342,A -85,B 0,C 180,E1 18355.041,E2 18355.041} C_VEL
LIN {X 0,Y 422.328,Z 837.468,A -85,B 0,C 180,E1 18361.056,E2 18361.056} C_VEL
LIN {X 0,Y 423.595,Z 840.435,A -85,B 0,C 180,E1 18369.535,E2 18369.535} C_VEL
LIN {X 0,Y 431.345,Z 853.3,A -85,B 0,C 180,E1 18377.619,E2 18377.619} C_VEL
LIN {X 0,Y 445.894,Z 880.227,A -85,B 0,C 180,E1 18386.398,E2 18386.398} C_VEL
LIN {X 0,Y 462.073,Z 919.93,A -85,B 0,C 180,E1 18394.453,E2 18394.453} C_VEL
LIN {X 0,Y 466.766,Z 940.935,A -85,B 0,C 180,E1 18397.514,E2 18397.514} C_VEL
LIN {X 0,Y 442.941,Z 1011.685,A -85,B 0,C 180,E1 18402.161,E2 18402.161} C_VEL
LIN {X 0,Y 416.354,Z 1074.223,A -85,B 0,C 180,E1 18408.94,E2 18408.94} C_VEL
LIN {X 0,Y 391.326,Z 1126.402,A -85,B 0,C 180,E1 18418.046,E2 18418.046} C_VEL
LIN {X 0,Y 373.303,Z 1165.639,A -85,B 0,C 180,E1 18429.276,E2 18429.276} C_VEL
LIN {X 0,Y 364.747,Z 1190.267,A -85,B 0,C 180,E1 18441.569,E2 18441.569} C_VEL
LIN {X 0,Y 363.071,Z 1199.409,A -85,B 0,C 180,E1 18451.138,E2 18451.138} C_VEL
LIN {X 0,Y 362.662,Z 1200.384,A -85,B 0,C 180,E1 18460.791,E2 18460.791} C_VEL
LIN {X 0,Y 364.655,Z 1191.31,A -85,B 0,C 180,E1 18471.929,E2 18471.929} C_VEL
LIN {X 0,Y 372.726,Z 1168.899,A -85,B 0,C 180,E1 18483.968,E2 18483.968} C_VEL
LIN {X 0,Y 391.595,Z 1130.647,A -85,B 0,C 180,E1 18495.712,E2 18495.712} C_VEL
LIN {X 0,Y 418.61,Z 1079.759,A -85,B 0,C 180,E1 18505.123,E2 18505.123} C_VEL
LIN {X 0,Y 447.325,Z 1019.567,A -85,B 0,C 180,E1 18511.98,E2 18511.98} C_VEL
LIN {X 0,Y 473.626,Z 951.025,A -85,B 0,C 180,E1 18516.704,E2 18516.704} C_VEL
LIN {X 0,Y 476.444,Z 938.983,A -85,B 0,C 180,E1 18517.556,E2 18517.556} C_VEL
LIN {X 0,Y 465.592,Z 905.52,A -85,B 0,C 180,E1 18525.093,E2 18525.093} C_VEL
LIN {X 0,Y 456.108,Z 882.81,A -85,B 0,C 180,E1 18533.41,E2 18533.41} C_VEL
LIN {X 0,Y 451.879,Z 875.508,A -85,B 0,C 180,E1 18540.456,E2 18540.456} C_VEL
LIN {X 0,Y 453.507,Z 878.634,A -85,B 0,C 180,E1 18549.92,E2 18549.92} C_VEL
LIN {X 0,Y 461.334,Z 894.961,A -85,B 0,C 180,E1 18558.176,E2 18558.176} C_VEL
LIN {X 0,Y 472.99,Z 924.111,A -85,B 0,C 180,E1 18566.14,E2 18566.14} C_VEL
LIN {X 0,Y 477.056,Z 943.181,A -85,B 0,C 180,E1 18569.474,E2 18569.474} C_VEL
LIN {X 0,Y 451.564,Z 1013.947,A -85,B 0,C 180,E1 18573.961,E2 18573.961} C_VEL
LIN {X 0,Y 422.529,Z 1076.64,A -85,B 0,C 180,E1 18580.484,E2 18580.484} C_VEL
LIN {X 0,Y 395.247,Z 1129.045,A -85,B 0,C 180,E1 18589.334,E2 18589.334} C_VEL
LIN {X 0,Y 375.454,Z 1168.849,A -85,B 0,C 180,E1 18600.242,E2 18600.242} C_VEL
LIN {X 0,Y 365.604,Z 1195.523,A -85,B 0,C 180,E1 18612.625,E2 18612.625} C_VEL
LIN {X 0,Y 363.19,Z 1207.377,A -85,B 0,C 180,E1 18624.064,E2 18624.064} C_VEL
LIN {X 0,Y 363.157,Z 1208.27,A -85,B 0,C 180,E1 18633.652,E2 18633.652} C_VEL
LIN {X 0,Y 364.349,Z 1199.13,A -85,B 0,C 180,E1 18644.53,E2 18644.53} C_VEL
LIN {X 0,Y 371.936,Z 1175.923,A -85,B 0,C 180,E1 18656.544,E2 18656.544} C_VEL
LIN {X 0,Y 388.548,Z 1137.747,A -85,B 0,C 180,E1 18667.91,E2 18667.91} C_VEL
LIN {X 0,Y 412.837,Z 1086.727,A -85,B 0,C 180,E1 18677.212,E2 18677.212} C_VEL
LIN {X 0,Y 431.667,Z 1044.263,A -85,B 0,C 180,E1 18682.373,E2 18682.373} C_VEL
LIN {X 0,Y 436.858,Z 1019.026,A -85,B 0,C 180,E1 18685.593,E2 18685.593} C_VEL
LIN {X 0,Y 461.727,Z 946.934,A -85,B 0,C 180,E1 18690.341,E2 18690.341} C_VEL
LIN {X 0,Y 462.535,Z 938.36,A -85,B 0,C 180,E1 18691.061,E2 18691.061} C_VEL
LIN {X 0,Y 447.848,Z 896.638,A -85,B 0,C 180,E1 18698.726,E2 18698.726} C_VEL
LIN {X 0,Y 431.778,Z 864.505,A -85,B 0,C 180,E1 18707.987,E2 18707.987} C_VEL
LIN {X 0,Y 423.286,Z 850.409,A -85,B 0,C 180,E1 18715.788,E2 18715.788} C_VEL
LIN {X 0,Y 420.817,Z 845.296,A -85,B 0,C 180,E1 18721.06,E2 18721.06} C_VEL
LIN {X 0,Y 422.001,Z 848.268,A -85,B 0,C 180,E1 18729.434,E2 18729.434} C_VEL
LIN {X 0,Y 429.442,Z 861.509,A -85,B 0,C 180,E1 18737.686,E2 18737.686} C_VEL
LIN {X 0,Y 443.365,Z 888.684,A -85,B 0,C 180,E1 18746.439,E2 18746.439} C_VEL
LIN {X 0,Y 457.896,Z 926.686,A -85,B 0,C 180,E1 18754.218,E2 18754.218} C_VEL
LIN {X 0,Y 461.608,Z 943.831,A -85,B 0,C 180,E1 18756.815,E2 18756.815} C_VEL
LIN {X 0,Y 436.658,Z 1015.052,A -85,B 0,C 180,E1 18761.589,E2 18761.589} C_VEL
LIN {X 0,Y 409.425,Z 1076.758,A -85,B 0,C 180,E1 18768.46,E2 18768.46} C_VEL
LIN {X 0,Y 383.87,Z 1128.067,A -85,B 0,C 180,E1 18777.685,E2 18777.685} C_VEL
LIN {X 0,Y 365.396,Z 1166.852,A -85,B 0,C 180,E1 18789.17,E2 18789.17} C_VEL
LIN {X 0,Y 356.824,Z 1190.498,A -85,B 0,C 180,E1 18801.38,E2 18801.38} C_VEL
LIN {X 0,Y 355.079,Z 1199.544,A -85,B 0,C 180,E1 18811.164,E2 18811.164} C_VEL
LIN {X 0,Y 354.655,Z 1200.423,A -85,B 0,C 180,E1 18821.038,E2 18821.038} C_VEL
LIN {X 0,Y 356.872,Z 1191.25,A -85,B 0,C 180,E1 18832.432,E2 18832.432} C_VEL
LIN {X 0,Y 365.369,Z 1168.94,A -85,B 0,C 180,E1 18844.64,E2 18844.64} C_VEL
LIN {X 0,Y 384.802,Z 1131.58,A -85,B 0,C 180,E1 18856.339,E2 18856.339} C_VEL
LIN {X 0,Y 412.421,Z 1081.548,A -85,B 0,C 180,E1 18865.777,E2 18865.777} C_VEL
LIN {X 0,Y 442.559,Z 1020.566,A -85,B 0,C 180,E1 18872.804,E2 18872.804} C_VEL
LIN {X 0,Y 469.989,Z 950.913,A -85,B 0,C 180,E1 18877.6,E2 18877.6} C_VEL
LIN {X 0,Y 471.308,Z 941.774,A -85,B 0,C 180,E1 18878.498,E2 18878.498} C_VEL
LIN {X 0,Y 461.176,Z 909.631,A -85,B 0,C 180,E1 18886.178,E2 18886.178} C_VEL
LIN {X 0,Y 453.784,Z 891.154,A -85,B 0,C 180,E1 18893.256,E2 18893.256} C_VEL
LIN {X 0,Y 449.667,Z 883.172,A -85,B 0,C 180,E1 18900.458,E2 18900.458} C_VEL
LIN {X 0,Y 451.239,Z 886.374,A -85,B 0,C 180,E1 18909.898,E2 18909.898} C_VEL
LIN {X 0,Y 458.687,Z 903.195,A -85,B 0,C 180,E1 18918.285,E2 18918.285} C_VEL
LIN {X 0,Y 469.423,Z 931.791,A -85,B 0,C 180,E1 18926.076,E2 18926.076} C_VEL
LIN {X 0,Y 472.08,Z 947.644,A -85,B 0,C 180,E1 18928.806,E2 18928.806} C_VEL
LIN {X 0,Y 445.117,Z 1019.023,A -85,B 0,C 180,E1 18933.458,E2 18933.458} C_VEL
LIN {X 0,Y 414.987,Z 1081.315,A -85,B 0,C 180,E1 18940.199,E2 18940.199} C_VEL
LIN {X 0,Y 386.211,Z 1134.291,A -85,B 0,C 180,E1 18949.665,E2 18949.665} C_VEL
LIN {X 0,Y 366.297,Z 1173.046,A -85,B 0,C 180,E1 18961.124,E2 18961.124} C_VEL
LIN {X 0,Y 357.318,Z 1197.114,A -85,B 0,C 180,E1 18973.269,E2 18973.269} C_VEL
LIN {X 0,Y 355.201,Z 1207.306,A -85,B 0,C 180,E1 18983.93,E2 18983.93} C_VEL
LIN {X 0,Y 355.159,Z 1208.166,A -85,B 0,C 180,E1 18993.735,E2 18993.735} C_VEL
LIN {X 0,Y 356.454,Z 1198.984,A -85,B 0,C 180,E1 19004.859,E2 19004.859} C_VEL
LIN {X 0,Y 364.622,Z 1175.115,A -85,B 0,C 180,E1 19017.372,E2 19017.372} C_VEL
LIN {X 0,Y 382.346,Z 1136.455,A -85,B 0,C 180,E1 19028.927,E2 19028.927} C_VEL
LIN {X 0,Y 407.66,Z 1085.297,A -85,B 0,C 180,E1 19038.226,E2 19038.226} C_VEL
LIN {X 0,Y 434.842,Z 1023.869,A -85,B 0,C 180,E1 19045.168,E2 19045.168} C_VEL
LIN {X 0,Y 436.858,Z 1019.026,A -85,B 0,C 180,E1 19045.593,E2 19045.593} C_VEL
LIN {X 0,Y 442.526,Z 991.962,A -85,B 0,C 180,E1 19048.498,E2 19048.498} C_VEL
LIN {X 0,Y 457.406,Z 942.847,A -85,B 0,C 180,E1 19051.625,E2 19051.625} C_VEL
LIN {X 0,Y 443.699,Z 902.143,A -85,B 0,C 180,E1 19059.33,E2 19059.33} C_VEL
LIN {X 0,Y 429.17,Z 871.647,A -85,B 0,C 180,E1 19068.394,E2 19068.394} C_VEL
LIN {X 0,Y 421.234,Z 857.989,A -85,B 0,C 180,E1 19076.059,E2 19076.059} C_VEL
LIN {X 0,Y 419.206,Z 853.12,A -85,B 0,C 180,E1 19081.064,E2 19081.064} C_VEL
LIN {X 0,Y 420.119,Z 855.921,A -85,B 0,C 180,E1 19089.248,E2 19089.248} C_VEL
LIN {X 0,Y 427.333,Z 869.308,A -85,B 0,C 180,E1 19097.59,E2 19097.59} C_VEL
LIN {X 0,Y 439.885,Z 895.417,A -85,B 0,C 180,E1 19106.113,E2 19106.113} C_VEL
LIN {X 0,Y 453.392,Z 932.909,A -85,B 0,C 180,E1 19113.924,E2 19113.924} C_VEL
LIN {X 0,Y 455.904,Z 948.373,A -85,B 0,C 180,E1 19116.203,E2 19116.203} C_VEL
LIN {X 0,Y 430.346,Z 1018.388,A -85,B 0,C 180,E1 19121.019,E2 19121.019} C_VEL
LIN {X 0,Y 402.423,Z 1079.366,A -85,B 0,C 180,E1 19127.989,E2 19127.989} C_VEL
LIN {X 0,Y 376.432,Z 1129.718,A -85,B 0,C 180,E1 19137.306,E2 19137.306} C_VEL
LIN {X 0,Y 357.732,Z 1167.441,A -85,B 0,C 180,E1 19148.804,E2 19148.804} C_VEL
LIN {X 0,Y 348.906,Z 1190.727,A -85,B 0,C 180,E1 19161.183,E2 19161.183} C_VEL
LIN {X 0,Y 347.075,Z 1199.679,A -85,B 0,C 180,E1 19171.191,E2 19171.191} C_VEL
LIN {X 0,Y 346.67,Z 1200.463,A -85,B 0,C 180,E1 19181.296,E2 19181.296} C_VEL
LIN {X 0,Y 349.082,Z 1191.195,A -85,B 0,C 180,E1 19192.961,E2 19192.961} C_VEL
LIN {X 0,Y 358.16,Z 1168.838,A -85,B 0,C 180,E1 19205.398,E2 19205.398} C_VEL
LIN {X 0,Y 378.38,Z 1131.916,A -85,B 0,C 180,E1 19217.138,E2 19217.138} C_VEL
LIN {X 0,Y 407.58,Z 1081.043,A -85,B 0,C 180,E1 19226.791,E2 19226.791} C_VEL
LIN {X 0,Y 438.696,Z 1019.836,A -85,B 0,C 180,E1 19233.801,E2 19233.801} C_VEL
LIN {X 0,Y 466.403,Z 951.005,A -85,B 0,C 180,E1 19238.498,E2 19238.498} C_VEL
LIN {X 0,Y 461.103,Z 925.984,A -85,B 0,C 180,E1 19243.736,E2 19243.736} C_VEL
LIN {X 0,Y 452.251,Z 901.611,A -85,B 0,C 180,E1 19251.9,E2 19251.9} C_VEL
LIN {X 0,Y 447.965,Z 891.278,A -85,B 0,C 180,E1 19259.004,E2 19259.004} C_VEL
LIN {X 0,Y 448.521,Z 892.059,A -85,B 0,C 180,E1 19268.728,E2 19268.728} C_VEL
LIN {X 0,Y 455.587,Z 910.135,A -85,B 0,C 180,E1 19277.976,E2 19277.976} C_VEL
LIN {X 0,Y 465.165,Z 937.739,A -85,B 0,C 180,E1 19285.677,E2 19285.677} C_VEL
LIN {X 0,Y 467.603,Z 950.453,A -85,B 0,C 180,E1 19288.048,E2 19288.048} C_VEL
LIN {X 0,Y 439.506,Z 1021.989,A -85,B 0,C 180,E1 19292.793,E2 19292.793} C_VEL
LIN {X 0,Y 408.563,Z 1083.574,A -85,B 0,C 180,E1 19299.601,E2 19299.601} C_VEL
LIN {X 0,Y 379.275,Z 1135.437,A -85,B 0,C 180,E1 19309.091,E2 19309.091} C_VEL
LIN {X 0,Y 358.458,Z 1174.21,A -85,B 0,C 180,E1 19320.94,E2 19320.94} C_VEL
LIN {X 0,Y 349.111,Z 1198.073,A -85,B 0,C 180,E1 19333.655,E2 19333.655} C_VEL
LIN {X 0,Y 347.198,Z 1207.235,A -85,B 0,C 180,E1 19343.79,E2 19343.79} C_VEL
LIN {X 0,Y 347.149,Z 1208.06,A -85,B 0,C 180,E1 19353.821,E2 19353.821} C_VEL
LIN {X 0,Y 348.581,Z 1198.838,A -85,B 0,C 180,E1 19365.203,E2 19365.203} C_VEL
LIN {X 0,Y 357.089,Z 1175.043,A -85,B 0,C 180,E1 19377.933,E2 19377.933} C_VEL
LIN {X 0,Y 375.637,Z 1136.472,A -85,B 0,C 180,E1 19389.657,E2 19389.657} C_VEL
LIN {X 0,Y 401.534,Z 1085.976,A -85,B 0,C 180,E1 19398.956,E2 19398.956} C_VEL
LIN {X 0,Y 429.537,Z 1024.597,A -85,B 0,C 180,E1 19405.963,E2 19405.963} C_VEL
LIN {X 0,Y 442.526,Z 991.962,A -85,B 0,C 180,E1 19408.498,E2 19408.498} C_VEL
LIN {X 0,Y 447.962,Z 963.62,A -85,B 0,C 180,E1 19411.159,E2 19411.159} C_VEL
LIN {X 0,Y 452.063,Z 946.431,A -85,B 0,C 180,E1 19412.354,E2 19412.354} C_VEL
LIN {X 0,Y 438.94,Z 905.962,A -85,B 0,C 180,E1 19420.336,E2 19420.336} C_VEL
LIN {X 0,Y 425.719,Z 877.713,A -85,B 0,C 180,E1 19429.245,E2 19429.245} C_VEL
LIN {X 0,Y 418.978,Z 865.187,A -85,B 0,C 180,E1 19436.622,E2 19436.622} C_VEL
LIN {X 0,Y 417.337,Z 860.897,A -85,B 0,C 180,E1 19441.069,E2 19441.069} C_VEL
LIN {X 0,Y 418.208,Z 863.778,A -85,B 0,C 180,E1 19449.224,E2 19449.224} C_VEL
LIN {X 0,Y 424.955,Z 877.158,A -85,B 0,C 180,E1 19457.555,E2 19457.555} C_VEL
LIN {X 0,Y 437.126,Z 903.844,A -85,B 0,C 180,E1 19466.214,E2 19466.214} C_VEL
LIN {X 0,Y 449.792,Z 942.234,A -85,B 0,C 180,E1 19474.179,E2 19474.179} C_VEL
LIN {X 0,Y 450.245,Z 952.803,A -85,B 0,C 180,E1 19475.567,E2 19475.567} C_VEL
LIN {X 0,Y 423.569,Z 1022.951,A -85,B 0,C 180,E1 19480.55,E2 19480.55} C_VEL
LIN {X 0,Y 394.849,Z 1083.111,A -85,B 0,C 180,E1 19487.669,E2 19487.669} C_VEL
LIN {X 0,Y 368.124,Z 1133.097,A -85,B 0,C 180,E1 19497.344,E2 19497.344} C_VEL
LIN {X 0,Y 349.116,Z 1170.218,A -85,B 0,C 180,E1 19509.335,E2 19509.335} C_VEL
LIN {X 0,Y 340.49,Z 1192.49,A -85,B 0,C 180,E1 19522.254,E2 19522.254} C_VEL
LIN {X 0,Y 339.042,Z 1200.831,A -85,B 0,C 180,E1 19533.786,E2 19533.786} C_VEL
LIN {X 0,Y 339.173,Z 1198.393,A -85,B 0,C 180,E1 19545.809,E2 19545.809} C_VEL
LIN {X 0,Y 343.691,Z 1184.371,A -85,B 0,C 180,E1 19558.3,E2 19558.3} C_VEL
LIN {X 0,Y 357.949,Z 1156.236,A -85,B 0,C 180,E1 19570.993,E2 19570.993} C_VEL
LIN {X 0,Y 383.854,Z 1112.879,A -85,B 0,C 180,E1 19582.3,E2 19582.3} C_VEL
LIN {X 0,Y 415.676,Z 1057.419,A -85,B 0,C 180,E1 19590.891,E2 19590.891} C_VEL
LIN {X 0,Y 446.243,Z 994.406,A -85,B 0,C 180,E1 19596.742,E2 19596.742} C_VEL
LIN {X 0,Y 462.008,Z 951.973,A -85,B 0,C 180,E1 19599.535,E2 19599.535} C_VEL
LIN {X 0,Y 453.507,Z 921.164,A -85,B 0,C 180,E1 19607.417,E2 19607.417} C_VEL
LIN {X 0,Y 447.587,Z 904.86,A -85,B 0,C 180,E1 19614.383,E2 19614.383} C_VEL
LIN {X 0,Y 444.694,Z 898.331,A -85,B 0,C 180,E1 19620.952,E2 19620.952} C_VEL
LIN {X 0,Y 446.156,Z 901.575,A -85,B 0,C 180,E1 19629.762,E2 19629.762} C_VEL
LIN {X 0,Y 453.107,Z 919.275,A -85,B 0,C 180,E1 19638.518,E2 19638.518} C_VEL
LIN {X 0,Y 462.165,Z 948.299,A -85,B 0,C 180,E1 19646.275,E2 19646.275} C_VEL
LIN {X 0,Y 462.493,Z 955.156,A -85,B 0,C 180,E1 19647.384,E2 19647.384} C_VEL
LIN {X 0,Y 433.348,Z 1026.178,A -85,B 0,C 180,E1 19652.221,E2 19652.221} C_VEL
LIN {X 0,Y 401.211,Z 1087.609,A -85,B 0,C 180,E1 19659.256,E2 19659.256} C_VEL
LIN {X 0,Y 370.844,Z 1139.177,A -85,B 0,C 180,E1 19669.131,E2 19669.131} C_VEL
LIN {X 0,Y 350.411,Z 1175.786,A -85,B 0,C 180,E1 19680.918,E2 19680.918} C_VEL
LIN {X 0,Y 341.276,Z 1198.045,A -85,B 0,C 180,E1 19693.269,E2 19693.269} C_VEL
LIN {X 0,Y 339.195,Z 1207.166,A -85,B 0,C 180,E1 19703.643,E2 19703.643} C_VEL
LIN {X 0,Y 339.155,Z 1207.954,A -85,B 0,C 180,E1 19713.911,E2 19713.911} C_VEL
LIN {X 0,Y 340.714,Z 1198.687,A -85,B 0,C 180,E1 19725.563,E2 19725.563} C_VEL
LIN {X 0,Y 349.675,Z 1174.817,A -85,B 0,C 180,E1 19738.579,E2 19738.579} C_VEL
LIN {X 0,Y 368.576,Z 1137.249,A -85,B 0,C 180,E1 19750.226,E2 19750.226} C_VEL
LIN {X 0,Y 395.916,Z 1085.741,A -85,B 0,C 180,E1 19759.848,E2 19759.848} C_VEL
LIN {X 0,Y 424.815,Z 1024.163,A -85,B 0,C 180,E1 19766.885,E2 19766.885} C_VEL
LIN {X 0,Y 447.962,Z 963.62,A -85,B 0,C 180,E1 19771.159,E2 19771.159} C_VEL
LIN {X 0,Y 448.154,Z 950.864,A -85,B 0,C 180,E1 19772.683,E2 19772.683} C_VEL
LIN {X 0,Y 444.396,Z 940.939,A -85,B 0,C 180,E1 19774.707,E2 19774.707} C_VEL
LIN {X 0,Y 432.204,Z 904.994,A -85,B 0,C 180,E1 19782.67,E2 19782.67} C_VEL
LIN {X 0,Y 420.599,Z 879.78,A -85,B 0,C 180,E1 19791.92,E2 19791.92} C_VEL
LIN {X 0,Y 415.474,Z 868.649,A -85,B 0,C 180,E1 19801.074,E2 19801.074} C_VEL
LIN {X 0,Y 416.184,Z 871.464,A -85,B 0,C 180,E1 19809.071,E2 19809.071} C_VEL
LIN {X 0,Y 422.483,Z 884.759,A -85,B 0,C 180,E1 19817.433,E2 19817.433} C_VEL
LIN {X 0,Y 434.075,Z 912.003,A -85,B 0,C 180,E1 19826.269,E2 19826.269} C_VEL
LIN {X 0,Y 445.524,Z 950.178,A -85,B 0,C 180,E1 19834.212,E2 19834.212} C_VEL
LIN {X 0,Y 442.082,Z 964.979,A -85,B 0,C 180,E1 19835.367,E2 19835.367} C_VEL
LIN {X 0,Y 414.703,Z 1032.26,A -85,B 0,C 180,E1 19840.529,E2 19840.529} C_VEL
LIN {X 0,Y 384.451,Z 1092.051,A -85,B 0,C 180,E1 19848.167,E2 19848.167} C_VEL
LIN {X 0,Y 357.852,Z 1139.796,A -85,B 0,C 180,E1 19858.282,E2 19858.282} C_VEL
LIN {X 0,Y 340.01,Z 1173.927,A -85,B 0,C 180,E1 19870.38,E2 19870.38} C_VEL
LIN {X 0,Y 332.15,Z 1194.223,A -85,B 0,C 180,E1 19883.378,E2 19883.378} C_VEL
LIN {X 0,Y 331.016,Z 1200.943,A -85,B 0,C 180,E1 19893.878,E2 19893.878} C_VEL
LIN {X 0,Y 330.964,Z 1199.468,A -85,B 0,C 180,E1 19904.537,E2 19904.537} C_VEL
LIN {X 0,Y 334.829,Z 1187.508,A -85,B 0,C 180,E1 19916.793,E2 19916.793} C_VEL
LIN {X 0,Y 347.845,Z 1161.705,A -85,B 0,C 180,E1 19929.831,E2 19929.831} C_VEL
LIN {X 0,Y 373.296,Z 1120.596,A -85,B 0,C 180,E1 19941.656,E2 19941.656} C_VEL
LIN {X 0,Y 406.105,Z 1066.503,A -85,B 0,C 180,E1 19950.748,E2 19950.748} C_VEL
LIN {X 0,Y 437.886,Z 1004.76,A -85,B 0,C 180,E1 19956.926,E2 19956.926} C_VEL
LIN {X 0,Y 457.078,Z 955.818,A -85,B 0,C 180,E1 19960.339,E2 19960.339} C_VEL
LIN {X 0,Y 449.528,Z 926.207,A -85,B 0,C 180,E1 19968.292,E2 19968.292} C_VEL
LIN {X 0,Y 444.332,Z 911.522,A -85,B 0,C 180,E1 19975.078,E2 19975.078} C_VEL
LIN {X 0,Y 442.13,Z 905.909,A -85,B 0,C 180,E1 19980.957,E2 19980.957} C_VEL
LIN {X 0,Y 443.292,Z 907.692,A -85,B 0,C 180,E1 19988.832,E2 19988.832} C_VEL
LIN {X 0,Y 449.622,Z 925.967,A -85,B 0,C 180,E1 19998.158,E2 19998.158} C_VEL
LIN {X 0,Y 457.785,Z 954.597,A -85,B 0,C 180,E1 20005.987,E2 20005.987} C_VEL
LIN {X 0,Y 456.783,Z 961.767,A -85,B 0,C 180,E1 20006.81,E2 20006.81} C_VEL
LIN {X 0,Y 427.249,Z 1030.353,A -85,B 0,C 180,E1 20011.633,E2 20011.633} C_VEL
LIN {X 0,Y 394.339,Z 1090.755,A -85,B 0,C 180,E1 20018.754,E2 20018.754} C_VEL
LIN {X 0,Y 364.107,Z 1140.066,A -85,B 0,C 180,E1 20028.457,E2 20028.457} C_VEL
LIN {X 0,Y 342.372,Z 1177.363,A -85,B 0,C 180,E1 20040.896,E2 20040.896} C_VEL
LIN {X 0,Y 332.863,Z 1199.594,A -85,B 0,C 180,E1 20054.195,E2 20054.195} C_VEL
LIN {X 0,Y 331.187,Z 1208.142,A -85,B 0,C 180,E1 20066.124,E2 20066.124} C_VEL
LIN {X 0,Y 331.165,Z 1206.797,A -85,B 0,C 180,E1 20076.642,E2 20076.642} C_VEL
LIN {X 0,Y 334.023,Z 1194.942,A -85,B 0,C 180,E1 20088.608,E2 20088.608} C_VEL
LIN {X 0,Y 344.64,Z 1169.621,A -85,B 0,C 180,E1 20101.235,E2 20101.235} C_VEL
LIN {X 0,Y 365.939,Z 1130.108,A -85,B 0,C 180,E1 20112.701,E2 20112.701} C_VEL
LIN {X 0,Y 394.045,Z 1078.499,A -85,B 0,C 180,E1 20121.766,E2 20121.766} C_VEL
LIN {X 0,Y 423.634,Z 1015.998,A -85,B 0,C 180,E1 20128.471,E2 20128.471} C_VEL
LIN {X 0,Y 447.176,Z 951.844,A -85,B 0,C 180,E1 20132.773,E2 20132.773} C_VEL
LIN {X 0,Y 444.396,Z 940.939,A -85,B 0,C 180,E1 20134.707,E2 20134.707} C_VEL
LIN {X 0,Y 434.671,Z 928.288,A -85,B 0,C 180,E1 20138.862,E2 20138.862} C_VEL
LIN {X 0,Y 423.377,Z 898.828,A -85,B 0,C 180,E1 20147.087,E2 20147.087} C_VEL
LIN {X 0,Y 415.335,Z 881.657,A -85,B 0,C 180,E1 20155.707,E2 20155.707} C_VEL
LIN {X 0,Y 413.348,Z 876.361,A -85,B 0,C 180,E1 20161.079,E2 20161.079} C_VEL
LIN {X 0,Y 413.945,Z 879.234,A -85,B 0,C 180,E1 20169.086,E2 20169.086} C_VEL
LIN {X 0,Y 419.902,Z 892.482,A -85,B 0,C 180,E1 20177.368,E2 20177.368} C_VEL
LIN {X 0,Y 430.599,Z 919.458,A -85,B 0,C 180,E1 20186.156,E2 20186.156} C_VEL
LIN {X 0,Y 440.474,Z 955.019,A -85,B 0,C 180,E1 20193.691,E2 20193.691} C_VEL
LIN {X 0,Y 413.437,Z 1024.498,A -85,B 0,C 180,E1 20198.85,E2 20198.85} C_VEL
LIN {X 0,Y 383.117,Z 1084.391,A -85,B 0,C 180,E1 20206.05,E2 20206.05} C_VEL
LIN {X 0,Y 354.857,Z 1133.521,A -85,B 0,C 180,E1 20215.789,E2 20215.789} C_VEL
LIN {X 0,Y 334.118,Z 1170.721,A -85,B 0,C 180,E1 20228.272,E2 20228.272} C_VEL
LIN {X 0,Y 324.636,Z 1192.936,A -85,B 0,C 180,E1 20241.873,E2 20241.873} C_VEL
LIN {X 0,Y 322.99,Z 1201.046,A -85,B 0,C 180,E1 20253.974,E2 20253.974} C_VEL
LIN {X 0,Y 323.064,Z 1199.052,A -85,B 0,C 180,E1 20265.593,E2 20265.593} C_VEL
LIN {X 0,Y 327.607,Z 1186.448,A -85,B 0,C 180,E1 20278.182,E2 20278.182} C_VEL
LIN {X 0,Y 342.841,Z 1158.964,A -85,B 0,C 180,E1 20291.725,E2 20291.725} C_VEL
LIN {X 0,Y 370.642,Z 1116.349,A -85,B 0,C 180,E1 20303.559,E2 20303.559} C_VEL
LIN {X 0,Y 404.089,Z 1062.382,A -85,B 0,C 180,E1 20312.29,E2 20312.29} C_VEL
LIN {X 0,Y 436.534,Z 999.962,A -85,B 0,C 180,E1 20318.265,E2 20318.265} C_VEL
LIN {X 0,Y 452.476,Z 960.948,A -85,B 0,C 180,E1 20320.882,E2 20320.882} C_VEL
LIN {X 0,Y 445.721,Z 932.274,A -85,B 0,C 180,E1 20328.806,E2 20328.806} C_VEL
LIN {X 0,Y 440.839,Z 917.846,A -85,B 0,C 180,E1 20336.028,E2 20336.028} C_VEL
LIN {X 0,Y 439.203,Z 912.944,A -85,B 0,C 180,E1 20342.944,E2 20342.944} C_VEL
LIN {X 0,Y 441.144,Z 918.247,A -85,B 0,C 180,E1 20350.875,E2 20350.875} C_VEL
LIN {X 0,Y 447.573,Z 937.623,A -85,B 0,C 180,E1 20359.545,E2 20359.545} C_VEL
LIN {X 0,Y 453.238,Z 962.507,A -85,B 0,C 180,E1 20365.91,E2 20365.91} C_VEL
LIN {X 0,Y 423.049,Z 1030.807,A -85,B 0,C 180,E1 20370.697,E2 20370.697} C_VEL
LIN {X 0,Y 389.431,Z 1090.688,A -85,B 0,C 180,E1 20377.755,E2 20377.755} C_VEL
LIN {X 0,Y 357.535,Z 1140.827,A -85,B 0,C 180,E1 20387.727,E2 20387.727} C_VEL
LIN {X 0,Y 335.11,Z 1177.417,A -85,B 0,C 180,E1 20400.203,E2 20400.203} C_VEL
LIN {X 0,Y 324.976,Z 1199.706,A -85,B 0,C 180,E1 20413.92,E2 20413.92} C_VEL
LIN {X 0,Y 323.174,Z 1208.067,A -85,B 0,C 180,E1 20426.028,E2 20426.028} C_VEL
LIN {X 0,Y 323.169,Z 1206.682,A -85,B 0,C 180,E1 20436.807,E2 20436.807} C_VEL
LIN {X 0,Y 326.202,Z 1194.769,A -85,B 0,C 180,E1 20449.071,E2 20449.071} C_VEL
LIN {X 0,Y 337.444,Z 1169.392,A -85,B 0,C 180,E1 20461.967,E2 20461.967} C_VEL
LIN {X 0,Y 360.007,Z 1129.276,A -85,B 0,C 180,E1 20473.723,E2 20473.723} C_VEL
LIN {X 0,Y 389.925,Z 1076.039,A -85,B 0,C 180,E1 20483.002,E2 20483.002} C_VEL
LIN {X 0,Y 420.501,Z 1012.604,A -85,B 0,C 180,E1 20489.656,E2 20489.656} C_VEL
LIN {X 0,Y 441.599,Z 954.265,A -85,B 0,C 180,E1 20493.711,E2 20493.711} C_VEL
LIN {X 0,Y 434.671,Z 928.288,A -85,B 0,C 180,E1 20498.862,E2 20498.862} C_VEL
LIN {X 0,Y 425.215,Z 918.638,A -85,B 0,C 180,E1 20503.263,E2 20503.263} C_VEL
LIN {X 0,Y 415.144,Z 894.07,A -85,B 0,C 180,E1 20512.68,E2 20512.68} C_VEL
LIN {X 0,Y 411.129,Z 884.048,A -85,B 0,C 180,E1 20521.085,E2 20521.085} C_VEL
LIN {X 0,Y 411.646,Z 886.825,A -85,B 0,C 180,E1 20528.933,E2 20528.933} C_VEL
LIN {X 0,Y 417.903,Z 901.485,A -85,B 0,C 180,E1 20538,E2 20538} C_VEL
LIN {X 0,Y 428.098,Z 930.26,A -85,B 0,C 180,E1 20546.889,E2 20546.889} C_VEL
LIN {X 0,Y 435.354,Z 961.025,A -85,B 0,C 180,E1 20553.291,E2 20553.291} C_VEL
LIN {X 0,Y 406.207,Z 1030.343,A -85,B 0,C 180,E1 20558.447,E2 20558.447} C_VEL
LIN {X 0,Y 374.481,Z 1090.11,A -85,B 0,C 180,E1 20565.985,E2 20565.985} C_VEL
LIN {X 0,Y 345.497,Z 1138.562,A -85,B 0,C 180,E1 20576.254,E2 20576.254} C_VEL
LIN {X 0,Y 325.89,Z 1172.62,A -85,B 0,C 180,E1 20588.444,E2 20588.444} C_VEL
LIN {X 0,Y 316.709,Z 1193.156,A -85,B 0,C 180,E1 20601.668,E2 20601.668} C_VEL
LIN {X 0,Y 314.961,Z 1201.148,A -85,B 0,C 180,E1 20614.076,E2 20614.076} C_VEL
LIN {X 0,Y 315.044,Z 1199.496,A -85,B 0,C 180,E1 20625.29,E2 20625.29} C_VEL
LIN {X 0,Y 319.857,Z 1186.788,A -85,B 0,C 180,E1 20638.598,E2 20638.598} C_VEL
LIN {X 0,Y 336.184,Z 1159.06,A -85,B 0,C 180,E1 20652.595,E2 20652.595} C_VEL
LIN {X 0,Y 364.135,Z 1117.93,A -85,B 0,C 180,E1 20664.242,E2 20664.242} C_VEL
LIN {X 0,Y 398.479,Z 1064.526,A -85,B 0,C 180,E1 20673.045,E2 20673.045} C_VEL
LIN {X 0,Y 431.74,Z 1002.697,A -85,B 0,C 180,E1 20679.043,E2 20679.043} C_VEL
LIN {X 0,Y 447.6,Z 964.879,A -85,B 0,C 180,E1 20681.704,E2 20681.704} C_VEL
LIN {X 0,Y 441.413,Z 936.314,A -85,B 0,C 180,E1 20690.08,E2 20690.08} C_VEL
LIN {X 0,Y 437.112,Z 921.453,A -85,B 0,C 180,E1 20698.98,E2 20698.98} C_VEL
LIN {X 0,Y 437.494,Z 923.032,A -85,B 0,C 180,E1 20708.95,E2 20708.95} C_VEL
LIN {X 0,Y 442.385,Z 939.391,A -85,B 0,C 180,E1 20717.536,E2 20717.536} C_VEL
LIN {X 0,Y 448.748,Z 965.857,A -85,B 0,C 180,E1 20725.101,E2 20725.101} C_VEL
LIN {X 0,Y 417.078,Z 1034.998,A -85,B 0,C 180,E1 20730.075,E2 20730.075} C_VEL
LIN {X 0,Y 381.759,Z 1095.313,A -85,B 0,C 180,E1 20737.45,E2 20737.45} C_VEL
LIN {X 0,Y 349.074,Z 1144.421,A -85,B 0,C 180,E1 20747.729,E2 20747.729} C_VEL
LIN {X 0,Y 326.333,Z 1180.326,A -85,B 0,C 180,E1 20760.853,E2 20760.853} C_VEL
LIN {X 0,Y 316.593,Z 1201.091,A -85,B 0,C 180,E1 20774.787,E2 20774.787} C_VEL
LIN {X 0,Y 315.161,Z 1207.99,A -85,B 0,C 180,E1 20785.927,E2 20785.927} C_VEL
LIN {X 0,Y 315.166,Z 1206.564,A -85,B 0,C 180,E1 20796.981,E2 20796.981} C_VEL
LIN {X 0,Y 318.388,Z 1194.592,A -85,B 0,C 180,E1 20809.558,E2 20809.558} C_VEL
LIN {X 0,Y 330.329,Z 1169.132,A -85,B 0,C 180,E1 20822.74,E2 20822.74} C_VEL
LIN {X 0,Y 353.899,Z 1128.908,A -85,B 0,C 180,E1 20834.676,E2 20834.676} C_VEL
LIN {X 0,Y 384.897,Z 1075.532,A -85,B 0,C 180,E1 20844.007,E2 20844.007} C_VEL
LIN {X 0,Y 416.084,Z 1012.54,A -85,B 0,C 180,E1 20850.593,E2 20850.593} C_VEL
LIN {X 0,Y 436.52,Z 958.883,A -85,B 0,C 180,E1 20854.283,E2 20854.283} C_VEL
LIN {X 0,Y 426.321,Z 921.6,A -85,B 0,C 180,E1 20862.423,E2 20862.423} C_VEL
LIN {X 0,Y 425.215,Z 918.638,A -85,B 0,C 180,E1 20863.263,E2 20863.263} C_VEL
LIN {X 0,Y 416.824,Z 912.359,A -85,B 0,C 180,E1 20867.902,E2 20867.902} C_VEL
LIN {X 0,Y 409.916,Z 895.832,A -85,B 0,C 180,E1 20876.846,E2 20876.846} C_VEL
LIN {X 0,Y 408.46,Z 891.695,A -85,B 0,C 180,E1 20883.221,E2 20883.221} C_VEL
LIN {X 0,Y 409.37,Z 895.373,A -85,B 0,C 180,E1 20889.627,E2 20889.627} C_VEL
LIN {X 0,Y 415.777,Z 911.291,A -85,B 0,C 180,E1 20898.777,E2 20898.777} C_VEL
LIN {X 0,Y 425.186,Z 940.812,A -85,B 0,C 180,E1 20907.569,E2 20907.569} C_VEL
LIN {X 0,Y 429.438,Z 966.51,A -85,B 0,C 180,E1 20912.669,E2 20912.669} C_VEL
LIN {X 0,Y 399.79,Z 1034.091,A -85,B 0,C 180,E1 20917.857,E2 20917.857} C_VEL
LIN {X 0,Y 367.754,Z 1092.253,A -85,B 0,C 180,E1 20925.38,E2 20925.38} C_VEL
LIN {X 0,Y 338.104,Z 1140.056,A -85,B 0,C 180,E1 20935.802,E2 20935.802} C_VEL
LIN {X 0,Y 317.28,Z 1174.86,A -85,B 0,C 180,E1 20948.91,E2 20948.91} C_VEL
LIN {X 0,Y 308.298,Z 1194.793,A -85,B 0,C 180,E1 20962.863,E2 20962.863} C_VEL
LIN {X 0,Y 306.941,Z 1201.25,A -85,B 0,C 180,E1 20974.182,E2 20974.182} C_VEL
LIN {X 0,Y 307.09,Z 1199.511,A -85,B 0,C 180,E1 20985.696,E2 20985.696} C_VEL
LIN {X 0,Y 312.35,Z 1186.713,A -85,B 0,C 180,E1 20999.351,E2 20999.351} C_VEL
LIN {X 0,Y 329.694,Z 1159.005,A -85,B 0,C 180,E1 21013.565,E2 21013.565} C_VEL
LIN {X 0,Y 359.107,Z 1117.581,A -85,B 0,C 180,E1 21025.372,E2 21025.372} C_VEL
LIN {X 0,Y 394.083,Z 1064.872,A -85,B 0,C 180,E1 21034.052,E2 21034.052} C_VEL
LIN {X 0,Y 427.647,Z 1004.169,A -85,B 0,C 180,E1 21039.94,E2 21039.94} C_VEL
LIN {X 0,Y 442.782,Z 969.284,A -85,B 0,C 180,E1 21042.418,E2 21042.418} C_VEL
LIN {X 0,Y 437.456,Z 941.492,A -85,B 0,C 180,E1 21050.996,E2 21050.996} C_VEL
LIN {X 0,Y 434.144,Z 928.928,A -85,B 0,C 180,E1 21058.973,E2 21058.973} C_VEL
LIN {X 0,Y 433.951,Z 928.865,A -85,B 0,C 180,E1 21067.001,E2 21067.001} C_VEL
LIN {X 0,Y 437.606,Z 942.054,A -85,B 0,C 180,E1 21075.625,E2 21075.625} C_VEL
LIN {X 0,Y 443.5,Z 967.428,A -85,B 0,C 180,E1 21083.691,E2 21083.691} C_VEL
LIN {X 0,Y 442.055,Z 974.85,A -85,B 0,C 180,E1 21084.671,E2 21084.671} C_VEL
LIN {X 0,Y 408.645,Z 1043.143,A -85,B 0,C 180,E1 21089.832,E2 21089.832} C_VEL
LIN {X 0,Y 372.523,Z 1101.883,A -85,B 0,C 180,E1 21097.512,E2 21097.512} C_VEL
LIN {X 0,Y 339.84,Z 1148.972,A -85,B 0,C 180,E1 21108.086,E2 21108.086} C_VEL
LIN {X 0,Y 317.838,Z 1182.538,A -85,B 0,C 180,E1 21121.273,E2 21121.273} C_VEL
LIN {X 0,Y 308.237,Z 1202.276,A -85,B 0,C 180,E1 21135.824,E2 21135.824} C_VEL
LIN {X 0,Y 307.156,Z 1207.91,A -85,B 0,C 180,E1 21145.821,E2 21145.821} C_VEL
LIN {X 0,Y 307.162,Z 1206.441,A -85,B 0,C 180,E1 21157.164,E2 21157.164} C_VEL
LIN {X 0,Y 310.607,Z 1194.414,A -85,B 0,C 180,E1 21170.069,E2 21170.069} C_VEL
LIN {X 0,Y 323.291,Z 1168.869,A -85,B 0,C 180,E1 21183.546,E2 21183.546} C_VEL
LIN {X 0,Y 347.974,Z 1128.541,A -85,B 0,C 180,E1 21195.649,E2 21195.649} C_VEL
LIN {X 0,Y 379.994,Z 1075.026,A -85,B 0,C 180,E1 21205.037,E2 21205.037} C_VEL
LIN {X 0,Y 412.44,Z 1011.021,A -85,B 0,C 180,E1 21211.664,E2 21211.664} C_VEL
LIN {X 0,Y 431.466,Z 963.419,A -85,B 0,C 180,E1 21214.883,E2 21214.883} C_VEL
LIN {X 0,Y 422.346,Z 927.479,A -85,B 0,C 180,E1 21222.971,E2 21222.971} C_VEL
LIN {X 0,Y 416.824,Z 912.359,A -85,B 0,C 180,E1 21227.902,E2 21227.902} C_VEL
LIN {X 0,Y 409.831,Z 909.317,A -85,B 0,C 180,E1 21232.73,E2 21232.73} C_VEL
LIN {X 0,Y 406.272,Z 899.312,A -85,B 0,C 180,E1 21241.098,E2 21241.098} C_VEL
LIN {X 0,Y 406.521,Z 901.57,A -85,B 0,C 180,E1 21248.504,E2 21248.504} C_VEL
LIN {X 0,Y 412.236,Z 917.664,A -85,B 0,C 180,E1 21258.256,E2 21258.256} C_VEL
LIN {X 0,Y 420.864,Z 946.776,A -85,B 0,C 180,E1 21267.142,E2 21267.142} C_VEL
LIN {X 0,Y 424.475,Z 969.536,A -85,B 0,C 180,E1 21271.894,E2 21271.894} C_VEL
LIN {X 0,Y 393.971,Z 1036.709,A -85,B 0,C 180,E1 21277.13,E2 21277.13} C_VEL
LIN {X 0,Y 360.065,Z 1095.959,A -85,B 0,C 180,E1 21285.02,E2 21285.02} C_VEL
LIN {X 0,Y 330.211,Z 1142.311,A -85,B 0,C 180,E1 21295.556,E2 21295.556} C_VEL
LIN {X 0,Y 308.922,Z 1176.611,A -85,B 0,C 180,E1 21309.145,E2 21309.145} C_VEL
LIN {X 0,Y 300.348,Z 1194.981,A -85,B 0,C 180,E1 21322.673,E2 21322.673} C_VEL
LIN {X 0,Y 298.912,Z 1201.353,A -85,B 0,C 180,E1 21334.295,E2 21334.295} C_VEL
LIN {X 0,Y 299.131,Z 1199.527,A -85,B 0,C 180,E1 21346.124,E2 21346.124} C_VEL
LIN {X 0,Y 304.934,Z 1186.621,A -85,B 0,C 180,E1 21360.153,E2 21360.153} C_VEL
LIN {X 0,Y 323.303,Z 1158.988,A -85,B 0,C 180,E1 21374.555,E2 21374.555} C_VEL
LIN {X 0,Y 354.219,Z 1117.238,A -85,B 0,C 180,E1 21386.534,E2 21386.534} C_VEL
LIN {X 0,Y 390.408,Z 1064.355,A -85,B 0,C 180,E1 21395.185,E2 21395.185} C_VEL
LIN {X 0,Y 424.793,Z 1003.398,A -85,B 0,C 180,E1 21401.022,E2 21401.022} C_VEL
LIN {X 0,Y 437.967,Z 973.586,A -85,B 0,C 180,E1 21403.195,E2 21403.195} C_VEL
LIN {X 0,Y 433.508,Z 946.793,A -85,B 0,C 180,E1 21411.927,E2 21411.927} C_VEL
LIN {X 0,Y 430.325,Z 935.6,A -85,B 0,C 180,E1 21420.983,E2 21420.983} C_VEL
LIN {X 0,Y 431.186,Z 938.147,A -85,B 0,C 180,E1 21429.082,E2 21429.082} C_VEL
LIN {X 0,Y 435.342,Z 954.794,A -85,B 0,C 180,E1 21437.725,E2 21437.725} C_VEL
LIN {X 0,Y 438.763,Z 975.528,A -85,B 0,C 180,E1 21443.718,E2 21443.718} C_VEL
LIN {X 0,Y 404.138,Z 1044.47,A -85,B 0,C 180,E1 21448.92,E2 21448.92} C_VEL
LIN {X 0,Y 367.552,Z 1102.136,A -85,B 0,C 180,E1 21456.491,E2 21456.491} C_VEL
LIN {X 0,Y 333.41,Z 1149.45,A -85,B 0,C 180,E1 21467.227,E2 21467.227} C_VEL
LIN {X 0,Y 310.615,Z 1182.4,A -85,B 0,C 180,E1 21480.433,E2 21480.433} C_VEL
LIN {X 0,Y 300.359,Z 1202.242,A -85,B 0,C 180,E1 21495.444,E2 21495.444} C_VEL
LIN {X 0,Y 298.975,Z 1208.185,A -85,B 0,C 180,E1 21508.618,E2 21508.618} C_VEL
LIN {X 0,Y 299.552,Z 1204.564,A -85,B 0,C 180,E1 21520.284,E2 21520.284} C_VEL
LIN {X 0,Y 304.856,Z 1189.636,A -85,B 0,C 180,E1 21533.8,E2 21533.8} C_VEL
LIN {X 0,Y 322.233,Z 1159.343,A -85,B 0,C 180,E1 21547.827,E2 21547.827} C_VEL
LIN {X 0,Y 350.34,Z 1115.475,A -85,B 0,C 180,E1 21559.373,E2 21559.373} C_VEL
LIN {X 0,Y 383.608,Z 1059.669,A -85,B 0,C 180,E1 21567.952,E2 21567.952} C_VEL
LIN {X 0,Y 415.628,Z 994.374,A -85,B 0,C 180,E1 21573.858,E2 21573.858} C_VEL
LIN {X 0,Y 426.107,Z 966.057,A -85,B 0,C 180,E1 21575.862,E2 21575.862} C_VEL
LIN {X 0,Y 417.901,Z 932.117,A -85,B 0,C 180,E1 21583.87,E2 21583.87} C_VEL
LIN {X 0,Y 409.831,Z 909.317,A -85,B 0,C 180,E1 21592.73,E2 21592.73} C_VEL
LIN {X 0,Y 404.373,Z 910.11,A -85,B 0,C 180,E1 21597.695,E2 21597.695} C_VEL
LIN {X 0,Y 403.504,Z 906.845,A -85,B 0,C 180,E1 21605.421,E2 21605.421} C_VEL
LIN {X 0,Y 406.944,Z 918.677,A -85,B 0,C 180,E1 21615.256,E2 21615.256} C_VEL
LIN {X 0,Y 414.221,Z 943.192,A -85,B 0,C 180,E1 21624.207,E2 21624.207} C_VEL
LIN {X 0,Y 419.33,Z 973.146,A -85,B 0,C 180,E1 21631.129,E2 21631.129} C_VEL
LIN {X 0,Y 388.184,Z 1039.387,A -85,B 0,C 180,E1 21636.389,E2 21636.389} C_VEL
LIN {X 0,Y 353.403,Z 1098.099,A -85,B 0,C 180,E1 21644.371,E2 21644.371} C_VEL
LIN {X 0,Y 322.533,Z 1144.284,A -85,B 0,C 180,E1 21655.215,E2 21655.215} C_VEL
LIN {X 0,Y 301.09,Z 1177.402,A -85,B 0,C 180,E1 21668.864,E2 21668.864} C_VEL
LIN {X 0,Y 292.403,Z 1195.167,A -85,B 0,C 180,E1 21682.472,E2 21682.472} C_VEL
LIN {X 0,Y 290.882,Z 1201.455,A -85,B 0,C 180,E1 21694.414,E2 21694.414} C_VEL
LIN {X 0,Y 291.192,Z 1199.545,A -85,B 0,C 180,E1 21706.577,E2 21706.577} C_VEL
LIN {X 0,Y 297.62,Z 1186.452,A -85,B 0,C 180,E1 21721.06,E2 21721.06} C_VEL
LIN {X 0,Y 317.46,Z 1158.459,A -85,B 0,C 180,E1 21735.786,E2 21735.786} C_VEL
LIN {X 0,Y 349.504,Z 1116.899,A -85,B 0,C 180,E1 21747.722,E2 21747.722} C_VEL
LIN {X 0,Y 387.145,Z 1063.404,A -85,B 0,C 180,E1 21756.404,E2 21756.404} C_VEL
LIN {X 0,Y 422.844,Z 1001.219,A -85,B 0,C 180,E1 21762.217,E2 21762.217} C_VEL
LIN {X 0,Y 433.23,Z 977.929,A -85,B 0,C 180,E1 21763.983,E2 21763.983} C_VEL
LIN {X 0,Y 429.604,Z 953.202,A -85,B 0,C 180,E1 21772.364,E2 21772.364} C_VEL
LIN {X 0,Y 427.093,Z 942.9,A -85,B 0,C 180,E1 21780.991,E2 21780.991} C_VEL
LIN {X 0,Y 427.913,Z 945.636,A -85,B 0,C 180,E1 21789.152,E2 21789.152} C_VEL
LIN {X 0,Y 431.653,Z 962.573,A -85,B 0,C 180,E1 21797.881,E2 21797.881} C_VEL
LIN {X 0,Y 433.917,Z 980.12,A -85,B 0,C 180,E1 21802.98,E2 21802.98} C_VEL
LIN {X 0,Y 398.592,Z 1047.72,A -85,B 0,C 180,E1 21808.17,E2 21808.17} C_VEL
LIN {X 0,Y 360.894,Z 1104.932,A -85,B 0,C 180,E1 21815.869,E2 21815.869} C_VEL
LIN {X 0,Y 325.613,Z 1151.941,A -85,B 0,C 180,E1 21826.951,E2 21826.951} C_VEL
LIN {X 0,Y 301.439,Z 1185.746,A -85,B 0,C 180,E1 21841.515,E2 21841.515} C_VEL
LIN {X 0,Y 292.041,Z 1203.429,A -85,B 0,C 180,E1 21856.555,E2 21856.555} C_VEL
LIN {X 0,Y 290.998,Z 1208.105,A -85,B 0,C 180,E1 21868.58,E2 21868.58} C_VEL
LIN {X 0,Y 291.569,Z 1204.436,A -85,B 0,C 180,E1 21880.569,E2 21880.569} C_VEL
LIN {X 0,Y 297.746,Z 1188.653,A -85,B 0,C 180,E1 21894.94,E2 21894.94} C_VEL
LIN {X 0,Y 317.042,Z 1157.053,A -85,B 0,C 180,E1 21909.441,E2 21909.441} C_VEL
LIN {X 0,Y 346.933,Z 1112.08,A -85,B 0,C 180,E1 21921.019,E2 21921.019} C_VEL
LIN {X 0,Y 381.094,Z 1055.784,A -85,B 0,C 180,E1 21929.414,E2 21929.414} C_VEL
LIN {X 0,Y 413.429,Z 990.299,A -85,B 0,C 180,E1 21935.13,E2 21935.13} C_VEL
LIN {X 0,Y 420.899,Z 969.605,A -85,B 0,C 180,E1 21936.674,E2 21936.674} C_VEL
LIN {X 0,Y 413.382,Z 936.712,A -85,B 0,C 180,E1 21944.815,E2 21944.815} C_VEL
LIN {X 0,Y 406.34,Z 915.383,A -85,B 0,C 180,E1 21953.598,E2 21953.598} C_VEL
LIN {X 0,Y 404.373,Z 910.11,A -85,B 0,C 180,E1 21957.695,E2 21957.695} C_VEL
LIN {X 0,Y 400.592,Z 914.349,A -85,B 0,C 180,E1 21962.724,E2 21962.724} C_VEL
LIN {X 0,Y 401.697,Z 919.362,A -85,B 0,C 180,E1 21970.913,E2 21970.913} C_VEL
LIN {X 0,Y 407.039,Z 937.519,A -85,B 0,C 180,E1 21980.003,E2 21980.003} C_VEL
LIN {X 0,Y 413.588,Z 967.685,A -85,B 0,C 180,E1 21988.509,E2 21988.509} C_VEL
LIN {X 0,Y 413.865,Z 977.75,A -85,B 0,C 180,E1 21990.409,E2 21990.409} C_VEL
LIN {X 0,Y 381.581,Z 1043.679,A -85,B 0,C 180,E1 21995.792,E2 21995.792} C_VEL
LIN {X 0,Y 346.036,Z 1101.364,A -85,B 0,C 180,E1 22003.896,E2 22003.896} C_VEL
LIN {X 0,Y 314.627,Z 1146.571,A -85,B 0,C 180,E1 22014.952,E2 22014.952} C_VEL
LIN {X 0,Y 292.562,Z 1179.358,A -85,B 0,C 180,E1 22029.223,E2 22029.223} C_VEL
LIN {X 0,Y 284.184,Z 1196.539,A -85,B 0,C 180,E1 22043.794,E2 22043.794} C_VEL
LIN {X 0,Y 282.662,Z 1201.781,A -85,B 0,C 180,E1 22056.519,E2 22056.519} C_VEL
LIN {X 0,Y 284.219,Z 1197.379,A -85,B 0,C 180,E1 22070.817,E2 22070.817} C_VEL
LIN {X 0,Y 294.607,Z 1180.168,A -85,B 0,C 180,E1 22086.228,E2 22086.228} C_VEL
LIN {X 0,Y 319.994,Z 1147.556,A -85,B 0,C 180,E1 22100.792,E2 22100.792} C_VEL
LIN {X 0,Y 356.024,Z 1102.059,A -85,B 0,C 180,E1 22111.801,E2 22111.801} C_VEL
LIN {X 0,Y 395.272,Z 1044.805,A -85,B 0,C 180,E1 22119.595,E2 22119.595} C_VEL
LIN {X 0,Y 428.579,Z 982.991,A -85,B 0,C 180,E1 22124.578,E2 22124.578} C_VEL
LIN {X 0,Y 425.723,Z 959.626,A -85,B 0,C 180,E1 22132.809,E2 22132.809} C_VEL
LIN {X 0,Y 423.697,Z 950.137,A -85,B 0,C 180,E1 22140.999,E2 22140.999} C_VEL
LIN {X 0,Y 424.384,Z 953.005,A -85,B 0,C 180,E1 22149.229,E2 22149.229} C_VEL
LIN {X 0,Y 427.712,Z 970.078,A -85,B 0,C 180,E1 22157.956,E2 22157.956} C_VEL
LIN {X 0,Y 429.235,Z 984.532,A -85,B 0,C 180,E1 22162.222,E2 22162.222} C_VEL
LIN {X 0,Y 392.742,Z 1051.601,A -85,B 0,C 180,E1 22167.483,E2 22167.483} C_VEL
LIN {X 0,Y 353.075,Z 1109.258,A -85,B 0,C 180,E1 22175.519,E2 22175.519} C_VEL
LIN {X 0,Y 317.083,Z 1155.144,A -85,B 0,C 180,E1 22186.956,E2 22186.956} C_VEL
LIN {X 0,Y 293.246,Z 1187.069,A -85,B 0,C 180,E1 22201.599,E2 22201.599} C_VEL
LIN {X 0,Y 284.133,Z 1203.397,A -85,B 0,C 180,E1 22216.173,E2 22216.173} C_VEL
LIN {X 0,Y 282.995,Z 1208.025,A -85,B 0,C 180,E1 22228.54,E2 22228.54} C_VEL
LIN {X 0,Y 283.605,Z 1204.307,A -85,B 0,C 180,E1 22240.869,E2 22240.869} C_VEL
LIN {X 0,Y 290.261,Z 1188.45,A -85,B 0,C 180,E1 22255.629,E2 22255.629} C_VEL
LIN {X 0,Y 310.584,Z 1156.757,A -85,B 0,C 180,E1 22270.428,E2 22270.428} C_VEL
LIN {X 0,Y 341.714,Z 1111.668,A -85,B 0,C 180,E1 22282.113,E2 22282.113} C_VEL
LIN {X 0,Y 376.768,Z 1055.417,A -85,B 0,C 180,E1 22290.492,E2 22290.492} C_VEL
LIN {X 0,Y 409.919,Z 989.717,A -85,B 0,C 180,E1 22296.166,E2 22296.166} C_VEL
LIN {X 0,Y 415.909,Z 974.616,A -85,B 0,C 180,E1 22297.194,E2 22297.194} C_VEL
LIN {X 0,Y 409.657,Z 943.715,A -85,B 0,C 180,E1 22305.006,E2 22305.006} C_VEL
LIN {X 0,Y 402.85,Z 921.167,A -85,B 0,C 180,E1 22314.627,E2 22314.627} C_VEL
LIN {X 0,Y 400.592,Z 914.349,A -85,B 0,C 180,E1 22322.724,E2 22322.724} C_VEL
LIN {X 0,Y 398,Z 923.244,A -85,B 0,C 180,E1 22327.672,E2 22327.672} C_VEL
LIN {X 0,Y 401.67,Z 937.796,A -85,B 0,C 180,E1 22337.149,E2 22337.149} C_VEL
LIN {X 0,Y 407.596,Z 964.766,A -85,B 0,C 180,E1 22345.963,E2 22345.963} C_VEL
LIN {X 0,Y 408.666,Z 981.712,A -85,B 0,C 180,E1 22349.627,E2 22349.627} C_VEL
LIN {X 0,Y 375.115,Z 1047.73,A -85,B 0,C 180,E1 22355.16,E2 22355.16} C_VEL
LIN {X 0,Y 338.159,Z 1105.285,A -85,B 0,C 180,E1 22363.565,E2 22363.565} C_VEL
LIN {X 0,Y 305.727,Z 1150.012,A -85,B 0,C 180,E1 22375.114,E2 22375.114} C_VEL
LIN {X 0,Y 283.98,Z 1181.105,A -85,B 0,C 180,E1 22389.598,E2 22389.598} C_VEL
LIN {X 0,Y 276.054,Z 1197.903,A -85,B 0,C 180,E1 22405.193,E2 22405.193} C_VEL
LIN {X 0,Y 274.6,Z 1202,A -85,B 0,C 180,E1 22417.861,E2 22417.861} C_VEL
LIN {X 0,Y 276.75,Z 1196.593,A -85,B 0,C 180,E1 22432.484,E2 22432.484} C_VEL
LIN {X 0,Y 288.767,Z 1178.314,A -85,B 0,C 180,E1 22448.311,E2 22448.311} C_VEL
LIN {X 0,Y 316.633,Z 1144.642,A -85,B 0,C 180,E1 22462.872,E2 22462.872} C_VEL
LIN {X 0,Y 354.484,Z 1098.324,A -85,B 0,C 180,E1 22473.624,E2 22473.624} C_VEL
LIN {X 0,Y 394.341,Z 1040.921,A -85,B 0,C 180,E1 22481.097,E2 22481.097} C_VEL
LIN {X 0,Y 423.802,Z 987.761,A -85,B 0,C 180,E1 22485.252,E2 22485.252} C_VEL
LIN {X 0,Y 421.632,Z 965.122,A -85,B 0,C 180,E1 22493.777,E2 22493.777} C_VEL
LIN {X 0,Y 420.136,Z 957.288,A -85,B 0,C 180,E1 22501.007,E2 22501.007} C_VEL
LIN {X 0,Y 420.794,Z 960.31,A -85,B 0,C 180,E1 22509.308,E2 22509.308} C_VEL
LIN {X 0,Y 423.467,Z 976.572,A -85,B 0,C 180,E1 22517.699,E2 22517.699} C_VEL
LIN {X 0,Y 424.189,Z 989.313,A -85,B 0,C 180,E1 22521.474,E2 22521.474} C_VEL
LIN {X 0,Y 386.854,Z 1055.299,A -85,B 0,C 180,E1 22526.771,E2 22526.771} C_VEL
LIN {X 0,Y 346.184,Z 1112.172,A -85,B 0,C 180,E1 22534.922,E2 22534.922} C_VEL
LIN {X 0,Y 309.165,Z 1157.499,A -85,B 0,C 180,E1 22546.697,E2 22546.697} C_VEL
LIN {X 0,Y 284.623,Z 1188.97,A -85,B 0,C 180,E1 22562.078,E2 22562.078} C_VEL
LIN {X 0,Y 276.227,Z 1203.366,A -85,B 0,C 180,E1 22575.769,E2 22575.769} C_VEL
LIN {X 0,Y 275.005,Z 1207.946,A -85,B 0,C 180,E1 22588.497,E2 22588.497} C_VEL
LIN {X 0,Y 275.632,Z 1204.177,A -85,B 0,C 180,E1 22601.188,E2 22601.188} C_VEL
LIN {X 0,Y 282.819,Z 1188.244,A -85,B 0,C 180,E1 22616.354,E2 22616.354} C_VEL
LIN {X 0,Y 304.165,Z 1156.537,A -85,B 0,C 180,E1 22631.428,E2 22631.428} C_VEL
LIN {X 0,Y 336.568,Z 1111.251,A -85,B 0,C 180,E1 22643.254,E2 22643.254} C_VEL
LIN {X 0,Y 373.2,Z 1054.029,A -85,B 0,C 180,E1 22651.708,E2 22651.708} C_VEL
LIN {X 0,Y 406.766,Z 988.634,A -85,B 0,C 180,E1 22657.256,E2 22657.256} C_VEL
LIN {X 0,Y 410.632,Z 977.175,A -85,B 0,C 180,E1 22658.265,E2 22658.265} C_VEL
LIN {X 0,Y 404.84,Z 946.858,A -85,B 0,C 180,E1 22666.485,E2 22666.485} C_VEL
LIN {X 0,Y 399.364,Z 927.28,A -85,B 0,C 180,E1 22675.672,E2 22675.672} C_VEL
LIN {X 0,Y 397.658,Z 921.769,A -85,B 0,C 180,E1 22683.309,E2 22683.309} C_VEL
LIN {X 0,Y 398,Z 923.244,A -85,B 0,C 180,E1 22687.672,E2 22687.672} C_VEL
LIN {X 0,Y 396.006,Z 936.367,A -85,B 0,C 180,E1 22692.439,E2 22692.439} C_VEL
LIN {X 0,Y 400.608,Z 956.774,A -85,B 0,C 180,E1 22701.47,E2 22701.47} C_VEL
LIN {X 0,Y 404.45,Z 983.272,A -85,B 0,C 180,E1 22708.666,E2 22708.666} C_VEL
LIN {X 0,Y 369.923,Z 1049.457,A -85,B 0,C 180,E1 22714.264,E2 22714.264} C_VEL
LIN {X 0,Y 332.618,Z 1105.809,A -85,B 0,C 180,E1 22722.55,E2 22722.55} C_VEL
LIN {X 0,Y 299.112,Z 1150.402,A -85,B 0,C 180,E1 22734.225,E2 22734.225} C_VEL
LIN {X 0,Y 276.457,Z 1181.373,A -85,B 0,C 180,E1 22749.017,E2 22749.017} C_VEL
LIN {X 0,Y 268.065,Z 1198.065,A -85,B 0,C 180,E1 22765.049,E2 22765.049} C_VEL
LIN {X 0,Y 266.584,Z 1202.081,A -85,B 0,C 180,E1 22778.099,E2 22778.099} C_VEL
LIN {X 0,Y 269.007,Z 1196.585,A -85,B 0,C 180,E1 22793.168,E2 22793.168} C_VEL
LIN {X 0,Y 281.663,Z 1178.585,A -85,B 0,C 180,E1 22809.17,E2 22809.17} C_VEL
LIN {X 0,Y 310.154,Z 1145.838,A -85,B 0,C 180,E1 22823.704,E2 22823.704} C_VEL
LIN {X 0,Y 349.652,Z 1099.252,A -85,B 0,C 180,E1 22834.672,E2 22834.672} C_VEL
LIN {X 0,Y 390.292,Z 1042.458,A -85,B 0,C 180,E1 22842.08,E2 22842.08} C_VEL
LIN {X 0,Y 419.064,Z 992.181,A -85,B 0,C 180,E1 22846.048,E2 22846.048} C_VEL
LIN {X 0,Y 417.655,Z 972.317,A -85,B 0,C 180,E1 22853.717,E2 22853.717} C_VEL
LIN {X 0,Y 416.579,Z 964.431,A -85,B 0,C 180,E1 22861.016,E2 22861.016} C_VEL
LIN {X 0,Y 417.099,Z 967.593,A -85,B 0,C 180,E1 22869.392,E2 22869.392} C_VEL
LIN {X 0,Y 419.355,Z 984.305,A -85,B 0,C 180,E1 22877.878,E2 22877.878} C_VEL
LIN {X 0,Y 419.222,Z 994.094,A -85,B 0,C 180,E1 22880.712,E2 22880.712} C_VEL
LIN {X 0,Y 380.848,Z 1059.273,A -85,B 0,C 180,E1 22886.068,E2 22886.068} C_VEL
LIN {X 0,Y 339.323,Z 1115.091,A -85,B 0,C 180,E1 22894.298,E2 22894.298} C_VEL
LIN {X 0,Y 303.102,Z 1157.62,A -85,B 0,C 180,E1 22905.607,E2 22905.607} C_VEL
LIN {X 0,Y 277.304,Z 1188.999,A -85,B 0,C 180,E1 22921.274,E2 22921.274} C_VEL
LIN {X 0,Y 268.353,Z 1203.337,A -85,B 0,C 180,E1 22935.343,E2 22935.343} C_VEL
LIN {X 0,Y 267.001,Z 1207.866,A -85,B 0,C 180,E1 22948.452,E2 22948.452} C_VEL
LIN {X 0,Y 267.676,Z 1204.047,A -85,B 0,C 180,E1 22961.525,E2 22961.525} C_VEL
LIN {X 0,Y 275.408,Z 1188.036,A -85,B 0,C 180,E1 22977.121,E2 22977.121} C_VEL
LIN {X 0,Y 297.765,Z 1156.413,A -85,B 0,C 180,E1 22992.437,E2 22992.437} C_VEL
LIN {X 0,Y 331.169,Z 1111.376,A -85,B 0,C 180,E1 23004.318,E2 23004.318} C_VEL
LIN {X 0,Y 367.88,Z 1055.765,A -85,B 0,C 180,E1 23012.592,E2 23012.592} C_VEL
LIN {X 0,Y 402.506,Z 990.25,A -85,B 0,C 180,E1 23018.185,E2 23018.185} C_VEL
LIN {X 0,Y 405.511,Z 980.481,A -85,B 0,C 180,E1 23019.214,E2 23019.214} C_VEL
LIN {X 0,Y 400.421,Z 951.649,A -85,B 0,C 180,E1 23027.448,E2 23027.448} C_VEL
LIN {X 0,Y 395.719,Z 933.504,A -85,B 0,C 180,E1 23036.733,E2 23036.733} C_VEL
LIN {X 0,Y 394.72,Z 929.193,A -85,B 0,C 180,E1 23043.334,E2 23043.334} C_VEL
LIN {X 0,Y 395.928,Z 935.983,A -85,B 0,C 180,E1 23052.194,E2 23052.194} C_VEL
LIN {X 0,Y 396.006,Z 936.367,A -85,B 0,C 180,E1 23052.439,E2 23052.439} C_VEL
LIN {X 0,Y 394.476,Z 952.462,A -85,B 0,C 180,E1 23057.048,E2 23057.048} C_VEL
LIN {X 0,Y 398.749,Z 979.63,A -85,B 0,C 180,E1 23065.976,E2 23065.976} C_VEL
LIN {X 0,Y 397.971,Z 990.229,A -85,B 0,C 180,E1 23068.097,E2 23068.097} C_VEL
LIN {X 0,Y 362.921,Z 1054.258,A -85,B 0,C 180,E1 23073.701,E2 23073.701} C_VEL
LIN {X 0,Y 323.979,Z 1110.607,A -85,B 0,C 180,E1 23082.374,E2 23082.374} C_VEL
LIN {X 0,Y 289.652,Z 1154.371,A -85,B 0,C 180,E1 23094.615,E2 23094.615} C_VEL
LIN {X 0,Y 267.05,Z 1184.32,A -85,B 0,C 180,E1 23110.314,E2 23110.314} C_VEL
LIN {X 0,Y 260.099,Z 1198.219,A -85,B 0,C 180,E1 23124.897,E2 23124.897} C_VEL
LIN {X 0,Y 258.546,Z 1202.155,A -85,B 0,C 180,E1 23138.353,E2 23138.353} C_VEL
LIN {X 0,Y 261.295,Z 1196.577,A -85,B 0,C 180,E1 23153.894,E2 23153.894} C_VEL
LIN {X 0,Y 274.819,Z 1178.586,A -85,B 0,C 180,E1 23170.245,E2 23170.245} C_VEL
LIN {X 0,Y 305.174,Z 1145.415,A -85,B 0,C 180,E1 23185.09,E2 23185.09} C_VEL
LIN {X 0,Y 345.964,Z 1098.89,A -85,B 0,C 180,E1 23195.973,E2 23195.973} C_VEL
LIN {X 0,Y 387.743,Z 1041.857,A -85,B 0,C 180,E1 23203.284,E2 23203.284} C_VEL
LIN {X 0,Y 414.395,Z 996.39,A -85,B 0,C 180,E1 23206.934,E2 23206.934} C_VEL
LIN {X 0,Y 413.417,Z 977.816,A -85,B 0,C 180,E1 23214.709,E2 23214.709} C_VEL
LIN {X 0,Y 412.722,Z 971.415,A -85,B 0,C 180,E1 23221.025,E2 23221.025} C_VEL
LIN {X 0,Y 413.163,Z 974.772,A -85,B 0,C 180,E1 23229.482,E2 23229.482} C_VEL
LIN {X 0,Y 414.928,Z 991.858,A -85,B 0,C 180,E1 23238.076,E2 23238.076} C_VEL
LIN {X 0,Y 414.083,Z 999.383,A -85,B 0,C 180,E1 23239.965,E2 23239.965} C_VEL
LIN {X 0,Y 374.405,Z 1063.968,A -85,B 0,C 180,E1 23245.416,E2 23245.416} C_VEL
LIN {X 0,Y 332.344,Z 1118.213,A -85,B 0,C 180,E1 23253.69,E2 23253.69} C_VEL
LIN {X 0,Y 293.861,Z 1161.609,A -85,B 0,C 180,E1 23265.912,E2 23265.912} C_VEL
LIN {X 0,Y 268.138,Z 1191.512,A -85,B 0,C 180,E1 23282.262,E2 23282.262} C_VEL
LIN {X 0,Y 259.625,Z 1205.137,A -85,B 0,C 180,E1 23298.282,E2 23298.282} C_VEL
LIN {X 0,Y 258.975,Z 1207.55,A -85,B 0,C 180,E1 23311.761,E2 23311.761} C_VEL
LIN {X 0,Y 260.96,Z 1200.587,A -85,B 0,C 180,E1 23326.59,E2 23326.59} C_VEL
LIN {X 0,Y 272.998,Z 1180.345,A -85,B 0,C 180,E1 23342.675,E2 23342.675} C_VEL
LIN {X 0,Y 300.083,Z 1145.031,A -85,B 0,C 180,E1 23357.256,E2 23357.256} C_VEL
LIN {X 0,Y 336.813,Z 1096.461,A -85,B 0,C 180,E1 23368.151,E2 23368.151} C_VEL
LIN {X 0,Y 375.059,Z 1036.685,A -85,B 0,C 180,E1 23375.674,E2 23375.674} C_VEL
LIN {X 0,Y 400.629,Z 985.516,A -85,B 0,C 180,E1 23379.778,E2 23379.778} C_VEL
LIN {X 0,Y 396.345,Z 957.888,A -85,B 0,C 180,E1 23387.878,E2 23387.878} C_VEL
LIN {X 0,Y 392.452,Z 940.89,A -85,B 0,C 180,E1 23396.705,E2 23396.705} C_VEL
LIN {X 0,Y 391.487,Z 936.502,A -85,B 0,C 180,E1 23403.361,E2 23403.361} C_VEL
LIN {X 0,Y 392.641,Z 943.572,A -85,B 0,C 180,E1 23412.298,E2 23412.298} C_VEL
LIN {X 0,Y 394.476,Z 952.462,A -85,B 0,C 180,E1 23417.048,E2 23417.048} C_VEL
LIN {X 0,Y 392.429,Z 971.449,A -85,B 0,C 180,E1 23421.438,E2 23421.438} C_VEL
LIN {X 0,Y 393.921,Z 991.965,A -85,B 0,C 180,E1 23427.13,E2 23427.13} C_VEL
LIN {X 0,Y 357.882,Z 1055.983,A -85,B 0,C 180,E1 23432.753,E2 23432.753} C_VEL
LIN {X 0,Y 318.589,Z 1111.13,A -85,B 0,C 180,E1 23441.3,E2 23441.3} C_VEL
LIN {X 0,Y 282.93,Z 1154.959,A -85,B 0,C 180,E1 23453.744,E2 23453.744} C_VEL
LIN {X 0,Y 259.295,Z 1184.857,A -85,B 0,C 180,E1 23469.916,E2 23469.916} C_VEL
LIN {X 0,Y 252.113,Z 1198.374,A -85,B 0,C 180,E1 23484.735,E2 23484.735} C_VEL
LIN {X 0,Y 250.509,Z 1202.23,A -85,B 0,C 180,E1 23498.623,E2 23498.623} C_VEL
LIN {X 0,Y 253.589,Z 1196.571,A -85,B 0,C 180,E1 23514.667,E2 23514.667} C_VEL
LIN {X 0,Y 268.162,Z 1178.536,A -85,B 0,C 180,E1 23531.402,E2 23531.402} C_VEL
LIN {X 0,Y 300.097,Z 1145.328,A -85,B 0,C 180,E1 23546.406,E2 23546.406} C_VEL
LIN {X 0,Y 342.746,Z 1098.225,A -85,B 0,C 180,E1 23557.341,E2 23557.341} C_VEL
LIN {X 0,Y 386.208,Z 1039.99,A -85,B 0,C 180,E1 23564.616,E2 23564.616} C_VEL
LIN {X 0,Y 409.669,Z 1001.204,A -85,B 0,C 180,E1 23567.65,E2 23567.65} C_VEL
LIN {X 0,Y 409.33,Z 984.893,A -85,B 0,C 180,E1 23574.656,E2 23574.656} C_VEL
LIN {X 0,Y 408.829,Z 978.417,A -85,B 0,C 180,E1 23581.035,E2 23581.035} C_VEL
LIN {X 0,Y 409.109,Z 980.717,A -85,B 0,C 180,E1 23588.501,E2 23588.501} C_VEL
LIN {X 0,Y 410.284,Z 996.454,A -85,B 0,C 180,E1 23597.175,E2 23597.175} C_VEL
LIN {X 0,Y 409.223,Z 1003.989,A -85,B 0,C 180,E1 23599.17,E2 23599.17} C_VEL
LIN {X 0,Y 368.629,Z 1067.547,A -85,B 0,C 180,E1 23604.634,E2 23604.634} C_VEL
LIN {X 0,Y 325.397,Z 1121.181,A -85,B 0,C 180,E1 23613.054,E2 23613.054} C_VEL
LIN {X 0,Y 286.461,Z 1163.201,A -85,B 0,C 180,E1 23625.362,E2 23625.362} C_VEL
LIN {X 0,Y 260.829,Z 1191.523,A -85,B 0,C 180,E1 23641.414,E2 23641.414} C_VEL
LIN {X 0,Y 251.673,Z 1205.091,A -85,B 0,C 180,E1 23657.906,E2 23657.906} C_VEL
LIN {X 0,Y 250.969,Z 1207.454,A -85,B 0,C 180,E1 23671.818,E2 23671.818} C_VEL
LIN {X 0,Y 253.124,Z 1200.436,A -85,B 0,C 180,E1 23687.12,E2 23687.12} C_VEL
LIN {X 0,Y 266.18,Z 1179.774,A -85,B 0,C 180,E1 23703.861,E2 23703.861} C_VEL
LIN {X 0,Y 294.369,Z 1144.693,A -85,B 0,C 180,E1 23718.473,E2 23718.473} C_VEL
LIN {X 0,Y 332.124,Z 1096.396,A -85,B 0,C 180,E1 23729.322,E2 23729.322} C_VEL
LIN {X 0,Y 371.707,Z 1036.055,A -85,B 0,C 180,E1 23736.843,E2 23736.843} C_VEL
LIN {X 0,Y 395.588,Z 989.802,A -85,B 0,C 180,E1 23740.503,E2 23740.503} C_VEL
LIN {X 0,Y 392.075,Z 963.116,A -85,B 0,C 180,E1 23748.718,E2 23748.718} C_VEL
LIN {X 0,Y 388.837,Z 947.126,A -85,B 0,C 180,E1 23757.794,E2 23757.794} C_VEL
LIN {X 0,Y 388.327,Z 944.081,A -85,B 0,C 180,E1 23765.634,E2 23765.634} C_VEL
LIN {X 0,Y 390.019,Z 956.141,A -85,B 0,C 180,E1 23775.306,E2 23775.306} C_VEL
LIN {X 0,Y 392.429,Z 971.449,A -85,B 0,C 180,E1 23781.438,E2 23781.438} C_VEL
LIN {X 0,Y 389.185,Z 992.731,A -85,B 0,C 180,E1 23785.611,E2 23785.611} C_VEL
LIN {X 0,Y 386.547,Z 1000.54,A -85,B 0,C 180,E1 23786.596,E2 23786.596} C_VEL
LIN {X 0,Y 349.148,Z 1063.414,A -85,B 0,C 180,E1 23792.441,E2 23792.441} C_VEL
LIN {X 0,Y 308.323,Z 1117.746,A -85,B 0,C 180,E1 23801.483,E2 23801.483} C_VEL
LIN {X 0,Y 273.173,Z 1159.002,A -85,B 0,C 180,E1 23814.228,E2 23814.228} C_VEL
LIN {X 0,Y 250.642,Z 1186.571,A -85,B 0,C 180,E1 23830.462,E2 23830.462} C_VEL
LIN {X 0,Y 244.139,Z 1198.528,A -85,B 0,C 180,E1 23844.563,E2 23844.563} C_VEL
LIN {X 0,Y 242.477,Z 1202.306,A -85,B 0,C 180,E1 23858.911,E2 23858.911} C_VEL
LIN {X 0,Y 245.796,Z 1196.753,A -85,B 0,C 180,E1 23875.203,E2 23875.203} C_VEL
LIN {X 0,Y 262.065,Z 1177.999,A -85,B 0,C 180,E1 23892.929,E2 23892.929} C_VEL
LIN {X 0,Y 295.313,Z 1145.077,A -85,B 0,C 180,E1 23907.831,E2 23907.831} C_VEL
LIN {X 0,Y 339.059,Z 1098.347,A -85,B 0,C 180,E1 23918.603,E2 23918.603} C_VEL
LIN {X 0,Y 383.174,Z 1040.665,A -85,B 0,C 180,E1 23925.734,E2 23925.734} C_VEL
LIN {X 0,Y 404.916,Z 1005.479,A -85,B 0,C 180,E1 23928.548,E2 23928.548} C_VEL
LIN {X 0,Y 404.915,Z 990.34,A -85,B 0,C 180,E1 23935.675,E2 23935.675} C_VEL
LIN {X 0,Y 404.794,Z 984.943,A -85,B 0,C 180,E1 23943.194,E2 23943.194} C_VEL
LIN {X 0,Y 405.127,Z 990.422,A -85,B 0,C 180,E1 23950.763,E2 23950.763} C_VEL
LIN {X 0,Y 405.753,Z 1005.985,A -85,B 0,C 180,E1 23958.157,E2 23958.157} C_VEL
LIN {X 0,Y 363.375,Z 1070.412,A -85,B 0,C 180,E1 23963.764,E2 23963.764} C_VEL
LIN {X 0,Y 318.417,Z 1124.094,A -85,B 0,C 180,E1 23972.405,E2 23972.405} C_VEL
LIN {X 0,Y 278.427,Z 1165.397,A -85,B 0,C 180,E1 23985.061,E2 23985.061} C_VEL
LIN {X 0,Y 252.615,Z 1192.559,A -85,B 0,C 180,E1 24001.438,E2 24001.438} C_VEL
LIN {X 0,Y 243.731,Z 1205.046,A -85,B 0,C 180,E1 24017.505,E2 24017.505} C_VEL
LIN {X 0,Y 243.001,Z 1207.629,A -85,B 0,C 180,E1 24028.299,E2 24028.299} C_VEL
LIN {X 0,Y 243.839,Z 1203.651,A -85,B 0,C 180,E1 24042.669,E2 24042.669} C_VEL
LIN {X 0,Y 253.931,Z 1186.88,A -85,B 0,C 180,E1 24060.069,E2 24060.069} C_VEL
LIN {X 0,Y 280.364,Z 1154.395,A -85,B 0,C 180,E1 24076.382,E2 24076.382} C_VEL
LIN {X 0,Y 318.434,Z 1108.382,A -85,B 0,C 180,E1 24088.382,E2 24088.382} C_VEL
LIN {X 0,Y 359.294,Z 1050.507,A -85,B 0,C 180,E1 24096.566,E2 24096.566} C_VEL
LIN {X 0,Y 390.539,Z 993.786,A -85,B 0,C 180,E1 24101.341,E2 24101.341} C_VEL
LIN {X 0,Y 387.851,Z 968.928,A -85,B 0,C 180,E1 24109.323,E2 24109.323} C_VEL
LIN {X 0,Y 385.256,Z 954.344,A -85,B 0,C 180,E1 24117.773,E2 24117.773} C_VEL
LIN {X 0,Y 384.853,Z 951.376,A -85,B 0,C 180,E1 24125.685,E2 24125.685} C_VEL
LIN {X 0,Y 386.42,Z 964.14,A -85,B 0,C 180,E1 24135.644,E2 24135.644} C_VEL
LIN {X 0,Y 388.886,Z 987.724,A -85,B 0,C 180,E1 24144.211,E2 24144.211} C_VEL
LIN {X 0,Y 389.185,Z 992.731,A -85,B 0,C 180,E1 24145.611,E2 24145.611} C_VEL
LIN {X 0,Y 384.467,Z 1001.871,A -85,B 0,C 180,E1 24146.194,E2 24146.194} C_VEL
LIN {X 0,Y 376.888,Z 1012.751,A -85,B 0,C 180,E1 24146.343,E2 24146.343} C_VEL
LIN {X 0,Y 336.911,Z 1075.308,A -85,B 0,C 180,E1 24152.771,E2 24152.771} C_VEL
LIN {X 0,Y 295.736,Z 1126.77,A -85,B 0,C 180,E1 24162.373,E2 24162.373} C_VEL
LIN {X 0,Y 260.398,Z 1166.139,A -85,B 0,C 180,E1 24176.291,E2 24176.291} C_VEL
LIN {X 0,Y 240.443,Z 1190.577,A -85,B 0,C 180,E1 24193.41,E2 24193.41} C_VEL
LIN {X 0,Y 235.436,Z 1200.469,A -85,B 0,C 180,E1 24208.249,E2 24208.249} C_VEL
LIN {X 0,Y 234.576,Z 1202.049,A -85,B 0,C 180,E1 24222.991,E2 24222.991} C_VEL
LIN {X 0,Y 240.494,Z 1193.811,A -85,B 0,C 180,E1 24240.172,E2 24240.172} C_VEL
LIN {X 0,Y 261.57,Z 1172.447,A -85,B 0,C 180,E1 24257.584,E2 24257.584} C_VEL
LIN {X 0,Y 300.211,Z 1135.621,A -85,B 0,C 180,E1 24272.032,E2 24272.032} C_VEL
LIN {X 0,Y 346.577,Z 1085.604,A -85,B 0,C 180,E1 24281.874,E2 24281.874} C_VEL
LIN {X 0,Y 390.369,Z 1026.299,A -85,B 0,C 180,E1 24288.09,E2 24288.09} C_VEL
LIN {X 0,Y 400.137,Z 1010.023,A -85,B 0,C 180,E1 24289.437,E2 24289.437} C_VEL
LIN {X 0,Y 400.548,Z 995.922,A -85,B 0,C 180,E1 24296.715,E2 24296.715} C_VEL
LIN {X 0,Y 400.601,Z 991.752,A -85,B 0,C 180,E1 24303.228,E2 24303.228} C_VEL
LIN {X 0,Y 400.831,Z 997.512,A -85,B 0,C 180,E1 24310.879,E2 24310.879} C_VEL
LIN {X 0,Y 400.506,Z 1011.444,A -85,B 0,C 180,E1 24317.412,E2 24317.412} C_VEL
LIN {X 0,Y 358.357,Z 1073.092,A -85,B 0,C 180,E1 24322.848,E2 24322.848} C_VEL
LIN {X 0,Y 312.637,Z 1125.79,A -85,B 0,C 180,E1 24331.456,E2 24331.456} C_VEL
LIN {X 0,Y 271.599,Z 1166.424,A -85,B 0,C 180,E1 24344.22,E2 24344.22} C_VEL
LIN {X 0,Y 245.248,Z 1192.703,A -85,B 0,C 180,E1 24360.636,E2 24360.636} C_VEL
LIN {X 0,Y 235.807,Z 1205.002,A -85,B 0,C 180,E1 24377.078,E2 24377.078} C_VEL
LIN {X 0,Y 235.001,Z 1207.55,A -85,B 0,C 180,E1 24388.241,E2 24388.241} C_VEL
LIN {X 0,Y 235.924,Z 1203.518,A -85,B 0,C 180,E1 24403.102,E2 24403.102} C_VEL
LIN {X 0,Y 246.464,Z 1186.979,A -85,B 0,C 180,E1 24420.803,E2 24420.803} C_VEL
LIN {X 0,Y 273.904,Z 1154.821,A -85,B 0,C 180,E1 24437.385,E2 24437.385} C_VEL
LIN {X 0,Y 313.111,Z 1109.118,A -85,B 0,C 180,E1 24449.465,E2 24449.465} C_VEL
LIN {X 0,Y 355.129,Z 1051.272,A -85,B 0,C 180,E1 24457.664,E2 24457.664} C_VEL
LIN {X 0,Y 385.585,Z 997.76,A -85,B 0,C 180,E1 24462.201,E2 24462.201} C_VEL
LIN {X 0,Y 383.426,Z 973.711,A -85,B 0,C 180,E1 24470.35,E2 24470.35} C_VEL
LIN {X 0,Y 381.525,Z 960.399,A -85,B 0,C 180,E1 24478.891,E2 24478.891} C_VEL
LIN {X 0,Y 381.261,Z 958.621,A -85,B 0,C 180,E1 24485.739,E2 24485.739} C_VEL
LIN {X 0,Y 382.224,Z 969.996,A -85,B 0,C 180,E1 24494.98,E2 24494.98} C_VEL
LIN {X 0,Y 384.067,Z 992.902,A -85,B 0,C 180,E1 24503.619,E2 24503.619} C_VEL
LIN {X 0,Y 383.128,Z 1001.249,A -85,B 0,C 180,E1 24505.518,E2 24505.518} C_VEL
LIN {X 0,Y 376.888,Z 1012.751,A -85,B 0,C 180,E1 24506.343,E2 24506.343} C_VEL
LIN {X 0,Y 356.779,Z 1040.92,A -85,B 0,C 180,E1 24507.567,E2 24507.567} C_VEL
LIN {X 0,Y 314.626,Z 1098.937,A -85,B 0,C 180,E1 24515.214,E2 24515.214} C_VEL
LIN {X 0,Y 273.737,Z 1145.33,A -85,B 0,C 180,E1 24526.584,E2 24526.584} C_VEL
LIN {X 0,Y 242.382,Z 1179.144,A -85,B 0,C 180,E1 24542.911,E2 24542.911} C_VEL
LIN {X 0,Y 229.055,Z 1196.622,A -85,B 0,C 180,E1 24560.373,E2 24560.373} C_VEL
LIN {X 0,Y 226.982,Z 1201.625,A -85,B 0,C 180,E1 24571.821,E2 24571.821} C_VEL
LIN {X 0,Y 227.12,Z 1201.158,A -85,B 0,C 180,E1 24587.396,E2 24587.396} C_VEL
LIN {X 0,Y 236.468,Z 1190.416,A -85,B 0,C 180,E1 24605.162,E2 24605.162} C_VEL
LIN {X 0,Y 264.407,Z 1164.766,A -85,B 0,C 180,E1 24622.904,E2 24622.904} C_VEL
LIN {X 0,Y 306.761,Z 1125.217,A -85,B 0,C 180,E1 24636.037,E2 24636.037} C_VEL
LIN {X 0,Y 353.536,Z 1073.816,A -85,B 0,C 180,E1 24644.704,E2 24644.704} C_VEL
LIN {X 0,Y 395.04,Z 1015.902,A -85,B 0,C 180,E1 24650.02,E2 24650.02} C_VEL
LIN {X 0,Y 396.16,Z 1002.722,A -85,B 0,C 180,E1 24656.678,E2 24656.678} C_VEL
LIN {X 0,Y 396.416,Z 998.547,A -85,B 0,C 180,E1 24663.262,E2 24663.262} C_VEL
LIN {X 0,Y 396.357,Z 1004.542,A -85,B 0,C 180,E1 24671.026,E2 24671.026} C_VEL
LIN {X 0,Y 395.428,Z 1016.644,A -85,B 0,C 180,E1 24676.6,E2 24676.6} C_VEL
LIN {X 0,Y 351.809,Z 1077.844,A -85,B 0,C 180,E1 24682.153,E2 24682.153} C_VEL
LIN {X 0,Y 305.415,Z 1129.047,A -85,B 0,C 180,E1 24690.814,E2 24690.814} C_VEL
LIN {X 0,Y 263.253,Z 1168.966,A -85,B 0,C 180,E1 24704.026,E2 24704.026} C_VEL
LIN {X 0,Y 236.334,Z 1194.457,A -85,B 0,C 180,E1 24721.32,E2 24721.32} C_VEL
LIN {X 0,Y 227.887,Z 1204.958,A -85,B 0,C 180,E1 24736.621,E2 24736.621} C_VEL
LIN {X 0,Y 226.995,Z 1207.471,A -85,B 0,C 180,E1 24748.179,E2 24748.179} C_VEL
LIN {X 0,Y 228.009,Z 1203.384,A -85,B 0,C 180,E1 24763.565,E2 24763.565} C_VEL
LIN {X 0,Y 239.07,Z 1187.064,A -85,B 0,C 180,E1 24781.592,E2 24781.592} C_VEL
LIN {X 0,Y 267.21,Z 1155.591,A -85,B 0,C 180,E1 24798.302,E2 24798.302} C_VEL
LIN {X 0,Y 307.624,Z 1110.181,A -85,B 0,C 180,E1 24810.519,E2 24810.519} C_VEL
LIN {X 0,Y 350.538,Z 1052.835,A -85,B 0,C 180,E1 24818.697,E2 24818.697} C_VEL
LIN {X 0,Y 380.688,Z 1001.191,A -85,B 0,C 180,E1 24823.24,E2 24823.24} C_VEL
LIN {X 0,Y 378.932,Z 977.402,A -85,B 0,C 180,E1 24831.976,E2 24831.976} C_VEL
LIN {X 0,Y 377.884,Z 965.685,A -85,B 0,C 180,E1 24841.18,E2 24841.18} C_VEL
LIN {X 0,Y 377.483,Z 967.588,A -85,B 0,C 180,E1 24848.116,E2 24848.116} C_VEL
LIN {X 0,Y 378.572,Z 981.25,A -85,B 0,C 180,E1 24856.92,E2 24856.92} C_VEL
LIN {X 0,Y 378.936,Z 1003.62,A -85,B 0,C 180,E1 24864.541,E2 24864.541} C_VEL
LIN {X 0,Y 356.779,Z 1040.92,A -85,B 0,C 180,E1 24867.567,E2 24867.567} C_VEL
LIN {X 0,Y 335.296,Z 1067.367,A -85,B 0,C 180,E1 24869.233,E2 24869.233} C_VEL
LIN {X 0,Y 290.909,Z 1121.235,A -85,B 0,C 180,E1 24878.406,E2 24878.406} C_VEL
LIN {X 0,Y 252.128,Z 1161.743,A -85,B 0,C 180,E1 24891.807,E2 24891.807} C_VEL
LIN {X 0,Y 227.525,Z 1187.815,A -85,B 0,C 180,E1 24908.975,E2 24908.975} C_VEL
LIN {X 0,Y 220.227,Z 1198.986,A -85,B 0,C 180,E1 24923.97,E2 24923.97} C_VEL
LIN {X 0,Y 218.64,Z 1202.368,A -85,B 0,C 180,E1 24935.876,E2 24935.876} C_VEL
LIN {X 0,Y 220.384,Z 1199.736,A -85,B 0,C 180,E1 24952.146,E2 24952.146} C_VEL
LIN {X 0,Y 234.97,Z 1185.27,A -85,B 0,C 180,E1 24971.321,E2 24971.321} C_VEL
LIN {X 0,Y 269.034,Z 1156.006,A -85,B 0,C 180,E1 24988.225,E2 24988.225} C_VEL
LIN {X 0,Y 315.67,Z 1112.688,A -85,B 0,C 180,E1 25000.113,E2 25000.113} C_VEL
LIN {X 0,Y 363.555,Z 1058.058,A -85,B 0,C 180,E1 25007.746,E2 25007.746} C_VEL
LIN {X 0,Y 390.627,Z 1019.621,A -85,B 0,C 180,E1 25011.035,E2 25011.035} C_VEL
LIN {X 0,Y 391.642,Z 1008.208,A -85,B 0,C 180,E1 25017.751,E2 25017.751} C_VEL
LIN {X 0,Y 391.993,Z 1005.757,A -85,B 0,C 180,E1 25025.523,E2 25025.523} C_VEL
LIN {X 0,Y 391.614,Z 1015.951,A -85,B 0,C 180,E1 25033.739,E2 25033.739} C_VEL
LIN {X 0,Y 390.104,Z 1021.98,A -85,B 0,C 180,E1 25035.8,E2 25035.8} C_VEL
LIN {X 0,Y 344.915,Z 1082.787,A -85,B 0,C 180,E1 25041.483,E2 25041.483} C_VEL
LIN {X 0,Y 296.259,Z 1133.998,A -85,B 0,C 180,E1 25050.597,E2 25050.597} C_VEL
LIN {X 0,Y 253.783,Z 1172.239,A -85,B 0,C 180,E1 25064.278,E2 25064.278} C_VEL
LIN {X 0,Y 227.294,Z 1196.271,A -85,B 0,C 180,E1 25082.249,E2 25082.249} C_VEL
LIN {X 0,Y 219.289,Z 1206.2,A -85,B 0,C 180,E1 25100.138,E2 25100.138} C_VEL
LIN {X 0,Y 218.967,Z 1207.068,A -85,B 0,C 180,E1 25112.083,E2 25112.083} C_VEL
LIN {X 0,Y 221.344,Z 1200.781,A -85,B 0,C 180,E1 25128.069,E2 25128.069} C_VEL
LIN {X 0,Y 237.049,Z 1180.912,A -85,B 0,C 180,E1 25146.958,E2 25146.958} C_VEL
LIN {X 0,Y 269.85,Z 1146.671,A -85,B 0,C 180,E1 25162.711,E2 25162.711} C_VEL
LIN {X 0,Y 312.901,Z 1098.484,A -85,B 0,C 180,E1 25173.931,E2 25173.931} C_VEL
LIN {X 0,Y 356.312,Z 1038.92,A -85,B 0,C 180,E1 25181.254,E2 25181.254} C_VEL
LIN {X 0,Y 375.694,Z 1005.929,A -85,B 0,C 180,E1 25183.9,E2 25183.9} C_VEL
LIN {X 0,Y 374.743,Z 983.262,A -85,B 0,C 180,E1 25192.635,E2 25192.635} C_VEL
LIN {X 0,Y 373.978,Z 972.712,A -85,B 0,C 180,E1 25201.193,E2 25201.193} C_VEL
LIN {X 0,Y 373.559,Z 974.714,A -85,B 0,C 180,E1 25208.202,E2 25208.202} C_VEL
LIN {X 0,Y 374.198,Z 989.576,A -85,B 0,C 180,E1 25217.473,E2 25217.473} C_VEL
LIN {X 0,Y 373.335,Z 1008.706,A -85,B 0,C 180,E1 25223.734,E2 25223.734} C_VEL
LIN {X 0,Y 335.296,Z 1067.367,A -85,B 0,C 180,E1 25229.233,E2 25229.233} C_VEL
LIN {X 0,Y 312.587,Z 1091.882,A -85,B 0,C 180,E1 25231.361,E2 25231.361} C_VEL
LIN {X 0,Y 268.571,Z 1139.778,A -85,B 0,C 180,E1 25242.023,E2 25242.023} C_VEL
LIN {X 0,Y 233.184,Z 1174.312,A -85,B 0,C 180,E1 25257.267,E2 25257.267} C_VEL
LIN {X 0,Y 215.085,Z 1194.357,A -85,B 0,C 180,E1 25275.603,E2 25275.603} C_VEL
LIN {X 0,Y 210.96,Z 1201.878,A -85,B 0,C 180,E1 25291.959,E2 25291.959} C_VEL
LIN {X 0,Y 211.358,Z 1201.259,A -85,B 0,C 180,E1 25308.74,E2 25308.74} C_VEL
LIN {X 0,Y 223.615,Z 1189.405,A -85,B 0,C 180,E1 25328.646,E2 25328.646} C_VEL
LIN {X 0,Y 257.001,Z 1162.009,A -85,B 0,C 180,E1 25347.194,E2 25347.194} C_VEL
LIN {X 0,Y 302.964,Z 1121.874,A -85,B 0,C 180,E1 25359.679,E2 25359.679} C_VEL
LIN {X 0,Y 352.195,Z 1069.474,A -85,B 0,C 180,E1 25367.819,E2 25367.819} C_VEL
LIN {X 0,Y 385.956,Z 1023.862,A -85,B 0,C 180,E1 25372.063,E2 25372.063} C_VEL
LIN {X 0,Y 387.277,Z 1013.69,A -85,B 0,C 180,E1 25378.848,E2 25378.848} C_VEL
LIN {X 0,Y 387.473,Z 1012.427,A -85,B 0,C 180,E1 25385.587,E2 25385.587} C_VEL
LIN {X 0,Y 386.733,Z 1022.253,A -85,B 0,C 180,E1 25393.582,E2 25393.582} C_VEL
LIN {X 0,Y 385.531,Z 1026.179,A -85,B 0,C 180,E1 25394.9,E2 25394.9} C_VEL
LIN {X 0,Y 339.798,Z 1085.581,A -85,B 0,C 180,E1 25400.513,E2 25400.513} C_VEL
LIN {X 0,Y 289.346,Z 1136.694,A -85,B 0,C 180,E1 25409.826,E2 25409.826} C_VEL
LIN {X 0,Y 246.107,Z 1173.869,A -85,B 0,C 180,E1 25423.723,E2 25423.723} C_VEL
LIN {X 0,Y 218.293,Z 1197.838,A -85,B 0,C 180,E1 25443.251,E2 25443.251} C_VEL
LIN {X 0,Y 211.309,Z 1206.138,A -85,B 0,C 180,E1 25459.762,E2 25459.762} C_VEL
LIN {X 0,Y 210.957,Z 1206.972,A -85,B 0,C 180,E1 25472.163,E2 25472.163} C_VEL
LIN {X 0,Y 213.589,Z 1200.627,A -85,B 0,C 180,E1 25488.749,E2 25488.749} C_VEL
LIN {X 0,Y 230.033,Z 1181.016,A -85,B 0,C 180,E1 25507.981,E2 25507.981} C_VEL
LIN {X 0,Y 264.783,Z 1146.322,A -85,B 0,C 180,E1 25524.175,E2 25524.175} C_VEL
LIN {X 0,Y 309.299,Z 1098.009,A -85,B 0,C 180,E1 25535.33,E2 25535.33} C_VEL
LIN {X 0,Y 353.291,Z 1038.901,A -85,B 0,C 180,E1 25542.481,E2 25542.481} C_VEL
LIN {X 0,Y 370.752,Z 1009.162,A -85,B 0,C 180,E1 25545.059,E2 25545.059} C_VEL
LIN {X 0,Y 370.332,Z 989.023,A -85,B 0,C 180,E1 25553.303,E2 25553.303} C_VEL
LIN {X 0,Y 370.068,Z 979.746,A -85,B 0,C 180,E1 25561.205,E2 25561.205} C_VEL
LIN {X 0,Y 369.605,Z 983.041,A -85,B 0,C 180,E1 25569.48,E2 25569.48} C_VEL
LIN {X 0,Y 369.788,Z 999.289,A -85,B 0,C 180,E1 25578.57,E2 25578.57} C_VEL
LIN {X 0,Y 368.18,Z 1013.115,A -85,B 0,C 180,E1 25582.85,E2 25582.85} C_VEL
LIN {X 0,Y 327.079,Z 1073.771,A -85,B 0,C 180,E1 25588.75,E2 25588.75} C_VEL
LIN {X 0,Y 312.587,Z 1091.882,A -85,B 0,C 180,E1 25591.361,E2 25591.361} C_VEL
LIN {X 0,Y 288.845,Z 1114.216,A -85,B 0,C 180,E1 25594.05,E2 25594.05} C_VEL
LIN {X 0,Y 245.378,Z 1157.248,A -85,B 0,C 180,E1 25607.023,E2 25607.023} C_VEL
LIN {X 0,Y 214.1,Z 1186.788,A -85,B 0,C 180,E1 25625.843,E2 25625.843} C_VEL
LIN {X 0,Y 204.314,Z 1199.289,A -85,B 0,C 180,E1 25643.499,E2 25643.499} C_VEL
LIN {X 0,Y 202.539,Z 1202.571,A -85,B 0,C 180,E1 25656.345,E2 25656.345} C_VEL
LIN {X 0,Y 204.943,Z 1199.786,A -85,B 0,C 180,E1 25673.914,E2 25673.914} C_VEL
LIN {X 0,Y 221.781,Z 1185.413,A -85,B 0,C 180,E1 25694.021,E2 25694.021} C_VEL
LIN {X 0,Y 259.231,Z 1156.378,A -85,B 0,C 180,E1 25711.223,E2 25711.223} C_VEL
LIN {X 0,Y 309.088,Z 1113.067,A -85,B 0,C 180,E1 25722.944,E2 25722.944} C_VEL
LIN {X 0,Y 359.171,Z 1058.445,A -85,B 0,C 180,E1 25730.282,E2 25730.282} C_VEL
LIN {X 0,Y 381.298,Z 1028.419,A -85,B 0,C 180,E1 25733.012,E2 25733.012} C_VEL
LIN {X 0,Y 382.85,Z 1018.776,A -85,B 0,C 180,E1 25741.105,E2 25741.105} C_VEL
LIN {X 0,Y 382.505,Z 1021.893,A -85,B 0,C 180,E1 25749.097,E2 25749.097} C_VEL
LIN {X 0,Y 380.709,Z 1030.919,A -85,B 0,C 180,E1 25754.028,E2 25754.028} C_VEL
LIN {X 0,Y 333.895,Z 1089.378,A -85,B 0,C 180,E1 25759.649,E2 25759.649} C_VEL
LIN {X 0,Y 283.186,Z 1138.755,A -85,B 0,C 180,E1 25768.847,E2 25768.847} C_VEL
LIN {X 0,Y 238.513,Z 1175.461,A -85,B 0,C 180,E1 25783.114,E2 25783.114} C_VEL
LIN {X 0,Y 210.955,Z 1197.835,A -85,B 0,C 180,E1 25802.242,E2 25802.242} C_VEL
LIN {X 0,Y 203.358,Z 1206.078,A -85,B 0,C 180,E1 25819.357,E2 25819.357} C_VEL
LIN {X 0,Y 202.947,Z 1206.875,A -85,B 0,C 180,E1 25832.248,E2 25832.248} C_VEL
LIN {X 0,Y 205.83,Z 1200.471,A -85,B 0,C 180,E1 25849.483,E2 25849.483} C_VEL
LIN {X 0,Y 223.104,Z 1181.12,A -85,B 0,C 180,E1 25869.064,E2 25869.064} C_VEL
LIN {X 0,Y 258.758,Z 1147.087,A -85,B 0,C 180,E1 25885.322,E2 25885.322} C_VEL
LIN {X 0,Y 304.359,Z 1099.266,A -85,B 0,C 180,E1 25896.477,E2 25896.477} C_VEL
LIN {X 0,Y 350.017,Z 1039.498,A -85,B 0,C 180,E1 25903.672,E2 25903.672} C_VEL
LIN {X 0,Y 365.823,Z 1014.435,A -85,B 0,C 180,E1 25905.602,E2 25905.602} C_VEL
LIN {X 0,Y 365.951,Z 994.617,A -85,B 0,C 180,E1 25914.083,E2 25914.083} C_VEL
LIN {X 0,Y 365.995,Z 986.668,A -85,B 0,C 180,E1 25921.219,E2 25921.219} C_VEL
LIN {X 0,Y 365.403,Z 988.841,A -85,B 0,C 180,E1 25928.386,E2 25928.386} C_VEL
LIN {X 0,Y 365.13,Z 1002.32,A -85,B 0,C 180,E1 25936.94,E2 25936.94} C_VEL
LIN {X 0,Y 363.931,Z 1016.07,A -85,B 0,C 180,E1 25941.844,E2 25941.844} C_VEL
LIN {X 0,Y 320.4,Z 1078.063,A -85,B 0,C 180,E1 25947.974,E2 25947.974} C_VEL
LIN {X 0,Y 288.845,Z 1114.216,A -85,B 0,C 180,E1 25954.05,E2 25954.05} C_VEL
LIN {X 0,Y 264.551,Z 1134.275,A -85,B 0,C 180,E1 25957.455,E2 25957.455} C_VEL
LIN {X 0,Y 224.303,Z 1170.718,A -85,B 0,C 180,E1 25972.377,E2 25972.377} C_VEL
LIN {X 0,Y 200.748,Z 1193.231,A -85,B 0,C 180,E1 25992.291,E2 25992.291} C_VEL
LIN {X 0,Y 195.56,Z 1201.102,A -85,B 0,C 180,E1 26007.667,E2 26007.667} C_VEL
LIN {X 0,Y 194.754,Z 1202.383,A -85,B 0,C 180,E1 26025.709,E2 26025.709} C_VEL
LIN {X 0,Y 205.334,Z 1193.124,A -85,B 0,C 180,E1 26046.96,E2 26046.96} C_VEL
LIN {X 0,Y 237.289,Z 1169.641,A -85,B 0,C 180,E1 26066.62,E2 26066.62} C_VEL
LIN {X 0,Y 285.047,Z 1132.074,A -85,B 0,C 180,E1 26080.386,E2 26080.386} C_VEL
LIN {X 0,Y 336.465,Z 1082.635,A -85,B 0,C 180,E1 26088.98,E2 26088.98} C_VEL
LIN {X 0,Y 376.552,Z 1033.426,A -85,B 0,C 180,E1 26093.782,E2 26093.782} C_VEL
LIN {X 0,Y 378.043,Z 1025.196,A -85,B 0,C 180,E1 26101.119,E2 26101.119} C_VEL
LIN {X 0,Y 377.605,Z 1028.521,A -85,B 0,C 180,E1 26109.218,E2 26109.218} C_VEL
LIN {X 0,Y 375.789,Z 1035.742,A -85,B 0,C 180,E1 26113.141,E2 26113.141} C_VEL
LIN {X 0,Y 327.105,Z 1094.158,A -85,B 0,C 180,E1 26118.895,E2 26118.895} C_VEL
LIN {X 0,Y 274.154,Z 1143.277,A -85,B 0,C 180,E1 26128.525,E2 26128.525} C_VEL
LIN {X 0,Y 227.421,Z 1179.582,A -85,B 0,C 180,E1 26144.096,E2 26144.096} C_VEL
LIN {X 0,Y 200.461,Z 1200.668,A -85,B 0,C 180,E1 26165.517,E2 26165.517} C_VEL
LIN {X 0,Y 195.074,Z 1206.795,A -85,B 0,C 180,E1 26183.411,E2 26183.411} C_VEL
